# B&R Automation Studio project Parker_BMM_ST_V5_3147_V12 (part 33)

#### nCarriageLR.apt
```
AcoposParameterTable:
  Root Parameters (Disabled=FALSE)
    Configure Parameter (Disabled=FALSE)
      128 = 1 (Name=SGEN_SW_END_IGNORE, Disabled=FALSE)  // Limit values: Ignore SW end positions
      1196 = 0 (Name=PCTRL_MODE_BITS, Disabled=FALSE)  // CTRL Position controller: Mode bits
      90 = 0 (Name=BRAKE_MODE, Disabled=FALSE)  // Motor holding brake: Mode
      80 = 1 (Name=PHASE_MON_IGNORE, Disabled=FALSE)  // Power mains: Ignore phase failure
      390 = 300 (Name=UDC_NOMINAL, Unit=V, Disabled=FALSE)  // CTRL DC bus: Nominal voltage
    VAR_XX_X+0 (Disabled=FALSE)
      777 = VAR_I4_0+0 (Name=FUNCTION_BLOCK_CREATE, Disabled=FALSE)  // VAR_XX_X+0
      VAR_R4_X_0 (Disabled=FALSE)
        4128 = 0.0 (Name=VAR_R4_0+0, Disabled=FALSE)  // velocity set -- cyclic set
        4136 = 0.0 (Name=VAR_R4_1+0, Disabled=FALSE)  // torque limit -- cyclic set
        4144 = 0.736 (Name=VAR_R4_2+0, Disabled=FALSE)  // temp junction Kp
        4152 = 0.736 (Name=VAR_R4_3+0, Disabled=FALSE)  // temp motor Kp
    VAR_XX_X+1 (Disabled=FALSE)
      777 = VAR_I4_0+1 (Name=FUNCTION_BLOCK_CREATE, Disabled=FALSE)  // VAR_XX_X+1
      VAR_R4_X_1 (Disabled=FALSE)
        4129 = 0.0 (Name=VAR_R4_0+1, Disabled=FALSE)  // zero
        4137 = 0.0 (Name=VAR_R4_1+1, Disabled=FALSE)  // 288 - SCTRL_ADD_SET_PARID
        4145 = 0.0 (Name=VAR_R4_2+1, Disabled=FALSE)  // no use
        4153 = 0.0 (Name=VAR_R4_3+1, Disabled=FALSE)  // no use
    VAR_XX_X+2 (Disabled=FALSE)
      777 = VAR_I4_0+2 (Name=FUNCTION_BLOCK_CREATE, Disabled=FALSE)  // VAR_XX_X+2
      VAR_R4_X_2 (Disabled=FALSE)
        4130 = 0.0 (Name=VAR_R4_0+2, Disabled=FALSE)  // Power Consumption Trigger - Left Carriage
        4138 = 0.0 (Name=VAR_R4_1+2, Disabled=FALSE)  // Power Consumption Trigger - Right Carriage
        4146 = 0.0 (Name=VAR_R4_2+2, Disabled=FALSE)  // FB2 FB VAR: Variable2 R4
        4154 = 0.0 (Name=VAR_R4_3+2, Disabled=FALSE)  // FB2 FB VAR: Variable3 R4
    VAR_XX_X+3 (Disabled=FALSE)
      777 = VAR_I4_0+3 (Name=FUNCTION_BLOCK_CREATE, Disabled=FALSE)  // VAR_XX_X+3
      VAR_R4_X_2 (Disabled=FALSE)
        4160 = 0.0 (Name=VAR_I2_0+0, Disabled=FALSE)  // FB0 FB VAR: Variable0 I2
        4168 = 0.0 (Name=VAR_I2_1+0, Disabled=FALSE)  // FB0 FB VAR: Variable1 I2
        4176 = 0.0 (Name=VAR_I2_2+0, Disabled=FALSE)  // FB0 FB VAR: Variable2 I2
        4184 = 0.0 (Name=VAR_I2_3+0, Disabled=FALSE)  // FB0 FB VAR: Variable3 I2
    Velocity Control (Disabled=FALSE)
      Function Create (Disabled=FALSE)
        777 = IPL_MODE+0 (Name=FUNCTION_BLOCK_CREATE, Disabled=FALSE)  // IPL_0
        777 = EVWR_MODE+0 (Name=FUNCTION_BLOCK_CREATE, Disabled=FALSE)  // EVWR_0
        777 = CMP_MODE+0 (Name=FUNCTION_BLOCK_CREATE, Disabled=FALSE)  // CMP_0
        777 = EVWR_MODE+1 (Name=FUNCTION_BLOCK_CREATE, Disabled=FALSE)  // EVWR_1
        777 = ARITH_MODE+6 (Name=FUNCTION_BLOCK_CREATE, Disabled=FALSE)  // EVWR_6
        777 = ARITH_MODE+7 (Name=FUNCTION_BLOCK_CREATE, Disabled=FALSE)  // EVWR_7
      IPL + 0 (Disabled=FALSE)
        8712 = VAR_R4_0+0 (Name=IPL_IN_PARID+0, Disabled=FALSE)  // velocity set
        8760 = CYCLIC_TODRV_COUNT (Name=IPL_EV_PARID+0, Disabled=FALSE)  // 909 - CYCLIC_TODRV_COUNT
        8720 = 2000 (Name=IPL_CYCLE_TIME+0, Unit=us, Disabled=FALSE)  // FB0 FB IPL: Cycle time
        8728 = 800 (Name=IPL_EXTRAPOLATION_TIME+0, Unit=us, Disabled=FALSE)  // FB0 FB IPL: Extrapolation time
        8704 = 1 (Name=IPL_MODE+0, Disabled=FALSE)  // linear interpolation
      EVWR + 0 (Disabled=FALSE)
        4608 = CMP_VALUE+0 (Name=EVWR_EVENT_PARID+0, Disabled=FALSE)  // v_set == 0
        4616 = IPL_VALUE_R4+0 (Name=EVWR_IN_PARID+0, Disabled=FALSE)  // 8752 -- interpolated v_set
        4624 = 0 (Name=EVWR_EVENT_LEVEL+0, Disabled=FALSE)  // FB0 FB EVWR: Event level
        4632 = VAR_R4_1+1 (Name=EVWR_WR_PARID+0, Disabled=FALSE)  // 288 - SCTRL_ADD_SET_PARID
        4640 = 2 (Name=EVWR_MODE+0, Disabled=FALSE)  // cyclic write
      ARITH + 6 (Disabled=FALSE)
        3598 = VCTRL_SCALE_LOAD_UNITS (Name=ARITH_IN1_PARID+6, Disabled=FALSE)  // FB6 FB ARITH: Parameter ID of input1
        3606 = VCTRL_SCALE_LOAD_MOTREV (Name=ARITH_IN2_PARID+6, Disabled=FALSE)  // FB6 FB ARITH: Parameter ID of input2
        3638 = 0 (Name=ARITH_K1+6, Disabled=FALSE)  // FB6 FB ARITH: Multiplication factor1
        3646 = 0 (Name=ARITH_K2+6, Disabled=FALSE)  // FB6 FB ARITH: Multiplication factor2
        3590 = 5 (Name=ARITH_MODE+6, Disabled=FALSE)  // FB6 FB ARITH: Mode
      ARITH + 7 (Disabled=FALSE)
        3599 = VAR_R4_1+1 (Name=ARITH_IN1_PARID+7, Disabled=FALSE)  // FB7 FB ARITH: Parameter ID of input1
        3607 = ARITH_VALUE_R4+6 (Name=ARITH_IN2_PARID+7, Disabled=FALSE)  // FB7 FB ARITH: Parameter ID of input2
        3639 = 0 (Name=ARITH_K1+7, Disabled=FALSE)  // FB7 FB ARITH: Multiplication factor1
        3647 = 0 (Name=ARITH_K2+7, Disabled=FALSE)  // FB7 FB ARITH: Multiplication factor2
        3591 = 5 (Name=ARITH_MODE+7, Disabled=FALSE)  // FB7 FB ARITH: Mode
      288 = ARITH_VALUE_R4+7 (Name=SCTRL_ADD_SET_PARID)  // CTRL Speed controller: Parameter ID additive set value
      CMP + 0 (Disabled=FALSE)
        6656 = IPL_VALUE_R4+0 (Name=CMP_IN_PARID+0, Disabled=FALSE)  // 8752 -- interpolated v_set
        6664 = 0 (Name=CMP_THRESHOLD+0, Disabled=FALSE)  // FB0 FB CMP: threshold
        6672 = 0.001 (Name=CMP_WINDOW+0, Disabled=FALSE)  // FB0 FB CMP: window
        6680 = 0 (Name=CMP_HYSTERESIS+0, Disabled=FALSE)  // FB0 FB CMP: hysteresis window
        6688 = 2 (Name=CMP_MODE+0, Disabled=FALSE)  // ==
      231 = CMP_VALUE+0 (Name=PCTRL_ENABLE_PARID, Disabled=FALSE)  // if(interpolated v_set == 0)enable PCTRL
      EVWR + 1 (Disabled=FALSE)
        4609 = CMP_VALUE+0 (Name=EVWR_EVENT_PARID+1, Disabled=FALSE)  // 6696
        4617 = MOTOR_TORQ_MAX (Name=EVWR_IN_PARID+1, Disabled=FALSE)  // FB1 FB EVWR: Parameter ID of input
        4625 = 1 (Name=EVWR_EVENT_LEVEL+1, Disabled=FALSE)  // FB1 FB EVWR: Event level
        4633 = VAR_R4_1+0 (Name=EVWR_WR_PARID+1, Disabled=FALSE)  // FB1 FB EVWR: Parameter ID of output value
        4641 = 2 (Name=EVWR_MODE+1, Disabled=FALSE)  // mode - cyclic write
    Torque Limitation (Disabled=FALSE)
      Function Create (Disabled=FALSE)
        777 = IPL_MODE+1 (Name=FUNCTION_BLOCK_CREATE, Disabled=FALSE)  // IPL_1
        777 = ARITH_MODE+0 (Name=FUNCTION_BLOCK_CREATE, Disabled=FALSE)  // ARITH_0
        777 = ARITH_MODE+1 (Name=FUNCTION_BLOCK_CREATE, Disabled=FALSE)  // ARITH_1
        777 = ARITH_MODE+2 (Name=FUNCTION_BLOCK_CREATE, Disabled=FALSE)  // ARITH_2
        777 = ARITH_MODE+3 (Name=FUNCTION_BLOCK_CREATE, Disabled=FALSE)  // ARITH_3
        777 = ARITH_MODE+4 (Name=FUNCTION_BLOCK_CREATE, Disabled=FALSE)  // ARITH_4
        777 = ARITH_MODE+5 (Name=FUNCTION_BLOCK_CREATE, Disabled=FALSE)  // ARITH_5
        777 = MINMAX_MODE+0 (Name=FUNCTION_BLOCK_CREATE, Disabled=FALSE)  // MINMAX_0
        777 = MINMAX_MODE+1 (Name=FUNCTION_BLOCK_CREATE, Disabled=FALSE)  // MINMAX_1
        777 = EVWR_MODE+2 (Name=FUNCTION_BLOCK_CREATE, Disabled=FALSE)  // EVWR_2
        777 = EVWR_MODE+3 (Name=FUNCTION_BLOCK_CREATE, Disabled=FALSE)  // EVWR_3
        777 = EVWR_MODE+4 (Name=FUNCTION_BLOCK_CREATE, Disabled=FALSE)  // EVWR_4
        777 = EVWR_MODE+5 (Name=FUNCTION_BLOCK_CREATE, Disabled=FALSE)  // EVWR_5
      IPL (Disabled=FALSE)
        8713 = VAR_R4_1+0 (Name=IPL_IN_PARID+1, Disabled=FALSE)  // 4136
        8761 = CYCLIC_TODRV_COUNT (Name=IPL_EV_PARID+1, Disabled=FALSE)  // 909 - CYCLIC_TODRV_COUNT
        8721 = 2000 (Name=IPL_CYCLE_TIME+1, Unit=us, Disabled=FALSE)  // FB1 FB IPL: Cycle time
        8729 = 2000 (Name=IPL_EXTRAPOLATION_TIME+1, Unit=us, Disabled=FALSE)  // FB1 FB IPL: Extrapolation time
        8705 = 1 (Name=IPL_MODE+1, Disabled=FALSE)  // FB1 FB IPL: Mode -- linear interpolation
      ARITH + 0 (Disabled=FALSE)
        3592 = TEMP_JUNCTION_LIM (Name=ARITH_IN1_PARID+0, Disabled=FALSE)  // TEMP_JUNCTION_LIM -- 842
        3600 = TEMP_JUNCTION (Name=ARITH_IN2_PARID+0, Disabled=FALSE)  // TEMP_JUNCTION -- 382
        3632 = 0 (Name=ARITH_K1+0, Disabled=FALSE)  // FB0 FB ARITH: Multiplication factor1
        3640 = 0 (Name=ARITH_K2+0, Disabled=FALSE)  // FB0 FB ARITH: Multiplication factor2
        3584 = 2 (Name=ARITH_MODE+0, Disabled=FALSE)  // y= x1 - x2
      ARITH + 1 (Disabled=FALSE)
        3593 = ARITH_VALUE_R4+0 (Name=ARITH_IN1_PARID+1, Disabled=FALSE)  // 3624
        3601 = VAR_R4_2+0 (Name=ARITH_IN2_PARID+1, Disabled=FALSE)  // 4144
        3633 = 0 (Name=ARITH_K1+1, Disabled=FALSE)  // FB1 FB ARITH: Multiplication factor1
        3641 = 0 (Name=ARITH_K2+1, Disabled=FALSE)  // FB1 FB ARITH: Multiplication factor2
        3585 = 3 (Name=ARITH_MODE+1, Disabled=FALSE)  // y = x1 * x2
      ARITH + 2 (Disabled=FALSE)
        3594 = MOTOR_TORQ_RATED (Name=ARITH_IN1_PARID+2, Disabled=FALSE)  // MOTOR_TORQ_RATED -- 53
        3602 = ARITH_VALUE_R4+1 (Name=ARITH_IN2_PARID+2, Disabled=FALSE)  // 3625
        3634 = 0 (Name=ARITH_K1+2, Disabled=FALSE)  // FB2 FB ARITH: Multiplication factor1
        3642 = 0 (Name=ARITH_K2+2, Disabled=FALSE)  // FB2 FB ARITH: Multiplication factor2
        3586 = 1 (Name=ARITH_MODE+2, Disabled=FALSE)  // y = x1 + x2
      ARITH + 3 (Disabled=FALSE)
        3595 = MOTOR_WIND_TEMP_MAX (Name=ARITH_IN1_PARID+3, Disabled=FALSE)  // 74 - MOTOR_WIND_TEMP_MAX
        3603 = TEMP_MOTOR_MODELL (Name=ARITH_IN2_PARID+3, Disabled=FALSE)  // 393 - TEMP_MOTOR_MODELL
        3635 = 0 (Name=ARITH_K1+3, Disabled=FALSE)  // FB3 FB ARITH: Multiplication factor1
        3643 = 0 (Name=ARITH_K2+3, Disabled=FALSE)  // FB3 FB ARITH: Multiplication factor2
        3587 = 2 (Name=ARITH_MODE+3, Disabled=FALSE)  // y = x1 - x2
      ARITH + 4 (Disabled=FALSE)
        3596 = ARITH_VALUE_R4+3 (Name=ARITH_IN1_PARID+4, Disabled=FALSE)  // 3627
        3604 = VAR_R4_3+0 (Name=ARITH_IN2_PARID+4, Disabled=FALSE)  // 4152
        3636 = 0 (Name=ARITH_K1+4, Disabled=FALSE)  // FB4 FB ARITH: Multiplication factor1
        3644 = 0 (Name=ARITH_K2+4, Disabled=FALSE)  // FB4 FB ARITH: Multiplication factor2
        3588 = 3 (Name=ARITH_MODE+4, Disabled=FALSE)  // y = x1 * x2
      ARITH + 5 (Disabled=FALSE)
        3597 = MOTOR_TORQ_RATED (Name=ARITH_IN1_PARID+5, Disabled=FALSE)  // MOTOR_TORQ_RATED -- 53
        3605 = ARITH_VALUE_R4+4 (Name=ARITH_IN2_PARID+5, Disabled=FALSE)  // 3628
        3637 = 0 (Name=ARITH_K1+5, Disabled=FALSE)  // FB5 FB ARITH: Multiplication factor1
        3645 = 0 (Name=ARITH_K2+5, Disabled=FALSE)  // FB5 FB ARITH: Multiplication factor2
        3589 = 1 (Name=ARITH_MODE+5, Disabled=FALSE)  // y = x1 + x2
      MINMAX + 0 (Disabled=FALSE)
        12312 = MOTOR_TORQ_MAX (Name=MINMAX_IN1_PARID+0, Disabled=FALSE)  // MOTOR_TORQ_MAX -- 54
        12320 = ARITH_VALUE_R4+2 (Name=MINMAX_IN2_PARID+0, Disabled=FALSE)  // 3626
        12328 = ARITH_VALUE_R4+5 (Name=MINMAX_IN3_PARID+0, Disabled=FALSE)  // 3629
        12336 = IPL_VALUE_R4+1 (Name=MINMAX_IN4_PARID+0, Disabled=FALSE)  // 8753 -- interpolated torque set
        12288 = 1 (Name=MINMAX_MODE+0, Disabled=FALSE)  // MIN(MOTOR_TORQ_MAX,ARITH_VALUE_R4+1)
      MINMAX + 1 (Disabled=FALSE)
        12313 = VAR_R4_0+1 (Name=MINMAX_IN1_PARID+1, Disabled=FALSE)  // zero
        12321 = MINMAX_VALUE_R4+0 (Name=MINMAX_IN2_PARID+1, Disabled=FALSE)  // FB1 FB MINMAX: Parameter ID of input2
        12289 = 2 (Name=MINMAX_MODE+1, Disabled=FALSE)  // MAX(VAR_R4_0+1,MINMAX_VALUE_R4+0)
      EVWR + 2 (Disabled=FALSE)
        4610 = CONST_I4_ONE (Name=EVWR_EVENT_PARID+2, Disabled=FALSE)  // FB2 FB EVWR: Parameter ID of event input
        4618 = MINMAX_VALUE_R4+1 (Name=EVWR_IN_PARID+2, Disabled=FALSE)  // FB2 FB EVWR: Parameter ID of input
        4626 = 1 (Name=EVWR_EVENT_LEVEL+2, Disabled=FALSE)  // FB2 FB EVWR: Event level
        4634 = LIM_T2_POS (Name=EVWR_WR_PARID+2, Disabled=FALSE)  // 348
        4642 = 2 (Name=EVWR_MODE+2, Disabled=FALSE)  // mode - cyclic write
      EVWR + 3 (Disabled=FALSE)
        4611 = CONST_I4_ONE (Name=EVWR_EVENT_PARID+3, Disabled=FALSE)  // FB3 FB EVWR: Parameter ID of event input
        4619 = MINMAX_VALUE_R4+1 (Name=EVWR_IN_PARID+3, Disabled=FALSE)  // FB3 FB EVWR: Parameter ID of input
        4627 = 1 (Name=EVWR_EVENT_LEVEL+3, Disabled=FALSE)  // FB3 FB EVWR: Event level
        4635 = LIM_T2_NEG (Name=EVWR_WR_PARID+3, Disabled=FALSE)  // 349
        4643 = 2 (Name=EVWR_MODE+3, Disabled=FALSE)  // mode - cyclic write
      EVWR + 4 (Disabled=FALSE)
        4612 = CONST_I4_ONE (Name=EVWR_EVENT_PARID+4, Disabled=FALSE)  // FB4 FB EVWR: Parameter ID of event input
        4620 = MINMAX_VALUE_R4+1 (Name=EVWR_IN_PARID+4, Disabled=FALSE)  // FB4 FB EVWR: Parameter ID of input
        4628 = 1 (Name=EVWR_EVENT_LEVEL+4, Disabled=FALSE)  // FB4 FB EVWR: Event level
        4636 = LIM_T1_POS (Name=EVWR_WR_PARID+4, Disabled=FALSE)  // 248
        4644 = 2 (Name=EVWR_MODE+4, Disabled=FALSE)  // mode - cyclic write
      EVWR + 5 (Disabled=FALSE)
        4613 = CONST_I4_ONE (Name=EVWR_EVENT_PARID+5, Disabled=FALSE)  // FB5 FB EVWR: Parameter ID of event input
        4621 = MINMAX_VALUE_R4+1 (Name=EVWR_IN_PARID+5, Disabled=FALSE)  // FB5 FB EVWR: Parameter ID of input
        4629 = 1 (Name=EVWR_EVENT_LEVEL+5, Disabled=FALSE)  // FB5 FB EVWR: Event level
        4637 = LIM_T1_NEG (Name=EVWR_WR_PARID+5, Disabled=FALSE)  // 249
        4645 = 2 (Name=EVWR_MODE+5, Disabled=FALSE)  // mode - cyclic write
    brake resistors (Disabled=TRUE)
      10 = 33 (Name=R_BLEEDER_EXT, Unit=Ohm, Disabled=TRUE)  // Bleeder: External: Resistance
      11 = 637 (Name=TEMP_MAX_BLEEDER_EXT, Unit=°C, Disabled=TRUE)  // Bleeder: External: Limit temperature
      12 = 0.852 (Name=RTH_BLEEDER_AMB_EXT, Unit=K/W, Disabled=TRUE)  // Bleeder: External: Thermal resistance
      13 = 40.68 (Name=CTH_BLEEDER_EXT, Unit=Ws/K, Disabled=TRUE)  // Bleeder: External: Thermal capacity
      398 = 1 (Name=BLEEDER_SELECTOR_EXT, Disabled=TRUE)  // Bleeder: Selector
    8B0W0079H000.000-1 mounting vertical V1 (Disabled=TRUE)
      brake  (Disabled=TRUE)  //  DO NOT USE with ACOPOS Firmware before V2.27.0
      10 = 33 (Name=R_BLEEDER_EXT, Unit=Ohm, Disabled=TRUE)  // Bleeder: External: Resistance
      11 = 673.08 (Name=TEMP_MAX_BLEEDER_EXT, Unit=癈, Disabled=TRUE)  // Bleeder: External: Limit temperature
      12 = 0.852 (Name=RTH_BLEEDER_AMB_EXT, Unit=K/W, Disabled=TRUE)  // Bleeder: External: Thermic resistance
      13 = 40.68 (Name=CTH_BLEEDER_EXT, Unit=Ws/K, Disabled=TRUE)  // Bleeder: External: Thermic capacity
      398 = 1 (Name=BLEEDER_SELECTOR_EXT, Disabled=TRUE)  // Bleeder: Selector
    Power Consumption (Disabled=TRUE)
      1140 = 10000000 (Name=PMET_TIME_IV, Unit=us, Disabled=TRUE)  // PowerMeter: Observation period
      1139 = 1 (Name=PMET_MODE, Disabled=TRUE)  // PowerMeter: Mode
    HardWare Limit  For ACOPOS Multi:
      945 = VAR_I2_0+0 (Name=POS_LIMIT_SWITCH_PARID)  // Digital inputs: Parameter ID for positive end switch
      946 = VAR_I2_1+0 (Name=NEG_LIMIT_SWITCH_PARID)  // Digital inputs: Parameter ID for negative end switch
```

### Data object Logical/Motion/para/BlowPin2LR (Apt)

#### BlowPin2LR.apt
```
AcoposParameterTable:
  Root Parameters (Disabled=FALSE)
    Configure Parameter (Disabled=FALSE)
      128 = 1 (Name=SGEN_SW_END_IGNORE, Disabled=FALSE)  // Limit values: Ignore SW end positions
      1196 = 0 (Name=PCTRL_MODE_BITS, Disabled=FALSE)  // CTRL Position controller: Mode bits
      80 = 1 (Name=PHASE_MON_IGNORE, Disabled=TRUE)  // Power mains: Ignore phase failure
      300 = 311 (Name=UDC_DETECTION, Unit=V, Disabled=FALSE)  // CTRL DC bus: Voltage detection: Lower limit
      373 = 1 (Name=TEMP_MOTOR_MODEL_MODE)  // Motor: Temperature model: Mode
      1215 = 2 (Name=MOTOR_TEMPSENS_TYPE, Disabled=TRUE)  // Temperature sensor: Type
    VAR_XX_X+0 (Disabled=FALSE)
      777 = VAR_I4_0+0 (Name=FUNCTION_BLOCK_CREATE, Disabled=FALSE)  // VAR_XX_X+0
      VAR_R4_X_0 (Disabled=FALSE)
        4128 = 0.0 (Name=VAR_R4_0+0, Disabled=FALSE)  // velocity set -- cyclic set
        4136 = 0.0 (Name=VAR_R4_1+0, Disabled=FALSE)  // torque limit -- cyclic set
        4144 = 0.666 (Name=VAR_R4_2+0, Disabled=FALSE)  // temp junction Kp
        4152 = 0.666 (Name=VAR_R4_3+0, Disabled=FALSE)  // temp motor Kp
    VAR_XX_X+1 (Disabled=FALSE)
      777 = VAR_I4_0+1 (Name=FUNCTION_BLOCK_CREATE, Disabled=FALSE)  // VAR_XX_X+1
      VAR_R4_X_1 (Disabled=FALSE)
        4129 = 0.0 (Name=VAR_R4_0+1, Disabled=FALSE)  // zero
        4137 = 0.0 (Name=VAR_R4_1+1, Disabled=FALSE)  // 288 - SCTRL_ADD_SET_PARID
        4145 = 0.0 (Name=VAR_R4_2+1, Disabled=FALSE)  // no use
        4153 = 0.0 (Name=VAR_R4_3+1, Disabled=FALSE)  // no use
    VAR_XX_X+3 (Disabled=FALSE)
      777 = VAR_I4_0+3 (Name=FUNCTION_BLOCK_CREATE, Disabled=FALSE)  // VAR_XX_X+3
      VAR_R4_X_2 (Disabled=FALSE)
        4160 = 0.0 (Name=VAR_I2_0+0, Disabled=FALSE)  // FB0 FB VAR: Variable0 I2
        4168 = 0.0 (Name=VAR_I2_1+0, Disabled=FALSE)  // FB0 FB VAR: Variable1 I2
        4176 = 0.0 (Name=VAR_I2_2+0, Disabled=FALSE)  // FB0 FB VAR: Variable2 I2
        4184 = 0.0 (Name=VAR_I2_3+0, Disabled=FALSE)  // FB0 FB VAR: Variable3 I2
    Velocity Control (Disabled=FALSE)
      Function Create (Disabled=FALSE)
        777 = IPL_MODE+0 (Name=FUNCTION_BLOCK_CREATE, Disabled=FALSE)  // IPL_0
        777 = EVWR_MODE+0 (Name=FUNCTION_BLOCK_CREATE, Disabled=FALSE)  // EVWR_0
        777 = CMP_MODE+0 (Name=FUNCTION_BLOCK_CREATE, Disabled=FALSE)  // CMP_0
        777 = EVWR_MODE+1 (Name=FUNCTION_BLOCK_CREATE, Disabled=FALSE)  // EVWR_1
      IPL + 0 (Disabled=FALSE)
        8712 = VAR_R4_0+0 (Name=IPL_IN_PARID+0, Disabled=FALSE)  // velocity set
        8760 = CYCLIC_TODRV_COUNT (Name=IPL_EV_PARID+0, Disabled=FALSE)  // 909 - CYCLIC_TODRV_COUNT
        8720 = 2000 (Name=IPL_CYCLE_TIME+0, Unit=us, Disabled=FALSE)  // FB0 FB IPL: Cycle time
        8728 = 800 (Name=IPL_EXTRAPOLATION_TIME+0, Unit=us, Disabled=FALSE)  // FB0 FB IPL: Extrapolation time
        8704 = 1 (Name=IPL_MODE+0, Disabled=FALSE)  // linear interpolation
      EVWR + 0 (Disabled=FALSE)
        4608 = CMP_VALUE+0 (Name=EVWR_EVENT_PARID+0, Disabled=FALSE)  // v_set == 0
        4616 = IPL_VALUE_R4+0 (Name=EVWR_IN_PARID+0, Disabled=FALSE)  // 8752 -- interpolated v_set
        4624 = 0 (Name=EVWR_EVENT_LEVEL+0, Disabled=FALSE)  // FB0 FB EVWR: Event level
        4632 = VAR_R4_1+1 (Name=EVWR_WR_PARID+0, Disabled=FALSE)  // 288-SCTRL_ADD_SET_PARID
        4640 = 2 (Name=EVWR_MODE+0, Disabled=FALSE)  // cyclic write
      288 = VAR_R4_1+1 (Name=SCTRL_ADD_SET_PARID, Disabled=FALSE)  // CTRL Speed controller: Parameter ID additive set value
      CMP + 0 (Disabled=FALSE)
        6656 = IPL_VALUE_R4+0 (Name=CMP_IN_PARID+0, Disabled=FALSE)  // 8752 -- interpolated v_set
        6664 = 0 (Name=CMP_THRESHOLD+0, Disabled=FALSE)  // FB0 FB CMP: threshold
        6672 = 0.001 (Name=CMP_WINDOW+0, Disabled=FALSE)  // FB0 FB CMP: window
        6680 = 0 (Name=CMP_HYSTERESIS+0, Disabled=FALSE)  // FB0 FB CMP: hysteresis window
        6688 = 2 (Name=CMP_MODE+0, Disabled=FALSE)  // ==
      231 = CMP_VALUE+0 (Name=PCTRL_ENABLE_PARID, Disabled=FALSE)  // if(interpolated v_set == 0)enable PCTRL
      EVWR + 1 (Disabled=FALSE)
        4609 = CMP_VALUE+0 (Name=EVWR_EVENT_PARID+1, Disabled=FALSE)  // 6696
        4617 = MOTOR_TORQ_MAX (Name=EVWR_IN_PARID+1, Disabled=FALSE)  // FB1 FB EVWR: Parameter ID of input
        4625 = 1 (Name=EVWR_EVENT_LEVEL+1, Disabled=FALSE)  // FB1 FB EVWR: Event level
        4633 = VAR_R4_1+0 (Name=EVWR_WR_PARID+1, Disabled=FALSE)  // FB1 FB EVWR: Parameter ID of output value
        4641 = 2 (Name=EVWR_MODE+1, Disabled=FALSE)  // mode - cyclic write
    Torque Limitation (Disabled=FALSE)
      Function Create (Disabled=FALSE)
        777 = IPL_MODE+1 (Name=FUNCTION_BLOCK_CREATE, Disabled=FALSE)  // IPL_1
        777 = ARITH_MODE+0 (Name=FUNCTION_BLOCK_CREATE, Disabled=FALSE)  // ARITH_0
        777 = ARITH_MODE+1 (Name=FUNCTION_BLOCK_CREATE, Disabled=FALSE)  // ARITH_1
        777 = ARITH_MODE+2 (Name=FUNCTION_BLOCK_CREATE, Disabled=FALSE)  // ARITH_2
        777 = ARITH_MODE+3 (Name=FUNCTION_BLOCK_CREATE, Disabled=FALSE)  // ARITH_3
        777 = ARITH_MODE+4 (Name=FUNCTION_BLOCK_CREATE, Disabled=FALSE)  // ARITH_4
        777 = ARITH_MODE+5 (Name=FUNCTION_BLOCK_CREATE, Disabled=FALSE)  // ARITH_5
        777 = MINMAX_MODE+0 (Name=FUNCTION_BLOCK_CREATE, Disabled=FALSE)  // MINMAX_0
        777 = MINMAX_MODE+1 (Name=FUNCTION_BLOCK_CREATE, Disabled=FALSE)  // MINMAX_1
        777 = EVWR_MODE+2 (Name=FUNCTION_BLOCK_CREATE, Disabled=FALSE)  // EVWR_2
        777 = EVWR_MODE+3 (Name=FUNCTION_BLOCK_CREATE, Disabled=FALSE)  // EVWR_3
        777 = EVWR_MODE+4 (Name=FUNCTION_BLOCK_CREATE, Disabled=FALSE)  // EVWR_4
        777 = EVWR_MODE+5 (Name=FUNCTION_BLOCK_CREATE, Disabled=FALSE)  // EVWR_5
      IPL (Disabled=FALSE)
        8713 = VAR_R4_1+0 (Name=IPL_IN_PARID+1, Disabled=FALSE)  // 4136
        8761 = CYCLIC_TODRV_COUNT (Name=IPL_EV_PARID+1, Disabled=FALSE)  // 909 - CYCLIC_TODRV_COUNT
        8721 = 2000 (Name=IPL_CYCLE_TIME+1, Unit=us, Disabled=FALSE)  // FB1 FB IPL: Cycle time
        8729 = 2000 (Name=IPL_EXTRAPOLATION_TIME+1, Unit=us, Disabled=FALSE)  // FB1 FB IPL: Extrapolation time
        8705 = 1 (Name=IPL_MODE+1, Disabled=FALSE)  // FB1 FB IPL: Mode -- linear interpolation
      ARITH + 0 (Disabled=FALSE)
        3592 = TEMP_JUNCTION_LIM (Name=ARITH_IN1_PARID+0, Disabled=FALSE)  // TEMP_JUNCTION_LIM -- 842
        3600 = TEMP_JUNCTION (Name=ARITH_IN2_PARID+0, Disabled=FALSE)  // TEMP_JUNCTION -- 382
        3632 = 0 (Name=ARITH_K1+0, Disabled=FALSE)  // FB0 FB ARITH: Multiplication factor1
        3640 = 0 (Name=ARITH_K2+0, Disabled=FALSE)  // FB0 FB ARITH: Multiplication factor2
        3584 = 2 (Name=ARITH_MODE+0, Disabled=FALSE)  // y= x1 - x2
      ARITH + 1 (Disabled=FALSE)
        3593 = ARITH_VALUE_R4+0 (Name=ARITH_IN1_PARID+1, Disabled=FALSE)  // 3624
        3601 = VAR_R4_2+0 (Name=ARITH_IN2_PARID+1, Disabled=FALSE)  // 4144
        3633 = 0 (Name=ARITH_K1+1, Disabled=FALSE)  // FB1 FB ARITH: Multiplication factor1
        3641 = 0 (Name=ARITH_K2+1, Disabled=FALSE)  // FB1 FB ARITH: Multiplication factor2
        3585 = 3 (Name=ARITH_MODE+1, Disabled=FALSE)  // y = x1 * x2
      ARITH + 2 (Disabled=FALSE)
        3594 = MOTOR_TORQ_RATED (Name=ARITH_IN1_PARID+2, Disabled=FALSE)  // MOTOR_TORQ_RATED -- 53
        3602 = ARITH_VALUE_R4+1 (Name=ARITH_IN2_PARID+2, Disabled=FALSE)  // 3625
        3634 = 0 (Name=ARITH_K1+2, Disabled=FALSE)  // FB2 FB ARITH: Multiplication factor1
        3642 = 0 (Name=ARITH_K2+2, Disabled=FALSE)  // FB2 FB ARITH: Multiplication factor2
        3586 = 1 (Name=ARITH_MODE+2, Disabled=FALSE)  // y = x1 + x2
      ARITH + 3 (Disabled=FALSE)
        3595 = MOTOR_WIND_TEMP_MAX (Name=ARITH_IN1_PARID+3, Disabled=FALSE)  // 74 - MOTOR_WIND_TEMP_MAX
        3603 = TEMP_MOTOR_MODELL (Name=ARITH_IN2_PARID+3, Disabled=FALSE)  // 393 - TEMP_MOTOR_MODELL
        3635 = 0 (Name=ARITH_K1+3, Disabled=FALSE)  // FB3 FB ARITH: Multiplication factor1
        3643 = 0 (Name=ARITH_K2+3, Disabled=FALSE)  // FB3 FB ARITH: Multiplication factor2
        3587 = 2 (Name=ARITH_MODE+3, Disabled=FALSE)  // y = x1 - x2
      ARITH + 4 (Disabled=FALSE)
        3596 = ARITH_VALUE_R4+3 (Name=ARITH_IN1_PARID+4, Disabled=FALSE)  // 3627
        3604 = VAR_R4_3+0 (Name=ARITH_IN2_PARID+4, Disabled=FALSE)  // 4152
        3636 = 0 (Name=ARITH_K1+4, Disabled=FALSE)  // FB4 FB ARITH: Multiplication factor1
        3644 = 0 (Name=ARITH_K2+4, Disabled=FALSE)  // FB4 FB ARITH: Multiplication factor2
        3588 = 3 (Name=ARITH_MODE+4, Disabled=FALSE)  // y = x1 * x2
      ARITH + 5 (Disabled=FALSE)
        3597 = MOTOR_TORQ_RATED (Name=ARITH_IN1_PARID+5, Disabled=FALSE)  // MOTOR_TORQ_RATED -- 53
        3605 = ARITH_VALUE_R4+4 (Name=ARITH_IN2_PARID+5, Disabled=FALSE)  // 3628
        3637 = 0 (Name=ARITH_K1+5, Disabled=FALSE)  // FB5 FB ARITH: Multiplication factor1
        3645 = 0 (Name=ARITH_K2+5, Disabled=FALSE)  // FB5 FB ARITH: Multiplication factor2
        3589 = 1 (Name=ARITH_MODE+5, Disabled=FALSE)  // y = x1 + x2
      MINMAX + 0 (Disabled=FALSE)
        12312 = MOTOR_TORQ_MAX (Name=MINMAX_IN1_PARID+0, Disabled=FALSE)  // MOTOR_TORQ_MAX -- 54
        12320 = ARITH_VALUE_R4+2 (Name=MINMAX_IN2_PARID+0, Disabled=FALSE)  // 3626
        12328 = ARITH_VALUE_R4+5 (Name=MINMAX_IN3_PARID+0, Disabled=FALSE)  // 3629
        12336 = IPL_VALUE_R4+1 (Name=MINMAX_IN4_PARID+0, Disabled=FALSE)  // 8753 -- interpolated torque set
        12288 = 1 (Name=MINMAX_MODE+0, Disabled=FALSE)  // MIN(MOTOR_TORQ_MAX,ARITH_VALUE_R4+1)
      MINMAX + 1 (Disabled=FALSE)
        12313 = VAR_R4_0+1 (Name=MINMAX_IN1_PARID+1, Disabled=FALSE)  // zero
        12321 = MINMAX_VALUE_R4+0 (Name=MINMAX_IN2_PARID+1, Disabled=FALSE)  // FB1 FB MINMAX: Parameter ID of input2
        12289 = 2 (Name=MINMAX_MODE+1, Disabled=FALSE)  // MAX(VAR_R4_0+1,MINMAX_VALUE_R4+0)
      EVWR + 2 (Disabled=FALSE)
        4610 = CONST_I4_ONE (Name=EVWR_EVENT_PARID+2, Disabled=FALSE)  // FB2 FB EVWR: Parameter ID of event input
        4618 = MINMAX_VALUE_R4+1 (Name=EVWR_IN_PARID+2, Disabled=FALSE)  // FB2 FB EVWR: Parameter ID of input
        4626 = 1 (Name=EVWR_EVENT_LEVEL+2, Disabled=FALSE)  // FB2 FB EVWR: Event level
        4634 = LIM_T2_POS (Name=EVWR_WR_PARID+2, Disabled=FALSE)  // 348
        4642 = 2 (Name=EVWR_MODE+2, Disabled=FALSE)  // mode - cyclic write
      EVWR + 3 (Disabled=FALSE)
        4611 = CONST_I4_ONE (Name=EVWR_EVENT_PARID+3, Disabled=FALSE)  // FB3 FB EVWR: Parameter ID of event input
        4619 = MINMAX_VALUE_R4+1 (Name=EVWR_IN_PARID+3, Disabled=FALSE)  // FB3 FB EVWR: Parameter ID of input
        4627 = 1 (Name=EVWR_EVENT_LEVEL+3, Disabled=FALSE)  // FB3 FB EVWR: Event level
        4635 = LIM_T2_NEG (Name=EVWR_WR_PARID+3, Disabled=FALSE)  // 349
        4643 = 2 (Name=EVWR_MODE+3, Disabled=FALSE)  // mode - cyclic write
      EVWR + 4 (Disabled=FALSE)
        4612 = CONST_I4_ONE (Name=EVWR_EVENT_PARID+4, Disabled=FALSE)  // FB4 FB EVWR: Parameter ID of event input
        4620 = MINMAX_VALUE_R4+1 (Name=EVWR_IN_PARID+4, Disabled=FALSE)  // FB4 FB EVWR: Parameter ID of input
        4628 = 1 (Name=EVWR_EVENT_LEVEL+4, Disabled=FALSE)  // FB4 FB EVWR: Event level
        4636 = LIM_T1_POS (Name=EVWR_WR_PARID+4, Disabled=FALSE)  // 248
        4644 = 2 (Name=EVWR_MODE+4, Disabled=FALSE)  // mode - cyclic write
      EVWR + 5 (Disabled=FALSE)
        4613 = CONST_I4_ONE (Name=EVWR_EVENT_PARID+5, Disabled=FALSE)  // FB5 FB EVWR: Parameter ID of event input
        4621 = MINMAX_VALUE_R4+1 (Name=EVWR_IN_PARID+5, Disabled=FALSE)  // FB5 FB EVWR: Parameter ID of input
        4629 = 1 (Name=EVWR_EVENT_LEVEL+5, Disabled=FALSE)  // FB5 FB EVWR: Event level
        4637 = LIM_T1_NEG (Name=EVWR_WR_PARID+5, Disabled=FALSE)  // 249
        4645 = 2 (Name=EVWR_MODE+5, Disabled=FALSE)  // mode - cyclic write
    HardWare Limit  For ACOPOS Multi:
      945 = VAR_I2_0+0 (Name=POS_LIMIT_SWITCH_PARID)  // Digital inputs: Parameter ID for positive end switch
      946 = VAR_I2_1+0 (Name=NEG_LIMIT_SWITCH_PARID)  // Digital inputs: Parameter ID for negative end switch
```

### Data object Logical/Motion/para/ClampLR (Apt)

#### ClampLR.apt
```
AcoposParameterTable:
  Root Parameters (Disabled=FALSE)
    Configure Parameter (Disabled=FALSE)
      128 = 1 (Name=SGEN_SW_END_IGNORE, Disabled=FALSE)  // Limit values: Ignore SW end positions
      1196 = 0 (Name=PCTRL_MODE_BITS, Disabled=FALSE)  // CTRL Position controller: Mode bits
      80 = 1 (Name=PHASE_MON_IGNORE, Disabled=FALSE)  // Power mains: Ignore phase failure
      300 = 300 (Name=UDC_DETECTION, Unit=V, Disabled=FALSE)  // CTRL DC bus: Voltage detection: Lower limit
      373 = 0 (Name=TEMP_MOTOR_MODEL_MODE)  // Motor: Temperature model: Mode
    VAR_XX_X+0 (Disabled=FALSE)
      777 = VAR_I4_0+0 (Name=FUNCTION_BLOCK_CREATE, Disabled=FALSE)  // VAR_XX_X+0
      VAR_R4_X_0 (Disabled=FALSE)
        4128 = 0.0 (Name=VAR_R4_0+0, Disabled=FALSE)  // velocity set -- cyclic set
        4136 = 0.0 (Name=VAR_R4_1+0, Disabled=FALSE)  // torque limit -- cyclic set
        4144 = 3.226 (Name=VAR_R4_2+0, Disabled=FALSE)  // temp junction Kp : (Peak - nominal)/50  (205-43.7)/50
        4152 = 3.226 (Name=VAR_R4_3+0, Disabled=FALSE)  // temp motor Kp
      VAR_I4_X_0 (Disabled=FALSE)
        4160 = 0.0 (Name=VAR_I2_0+0, Disabled=FALSE)  // FB0 FB VAR: Variable0 I2
        4168 = 0.0 (Name=VAR_I2_1+0, Disabled=FALSE)  // FB0 FB VAR: Variable1 I2
        4176 = 0.0 (Name=VAR_I2_2+0, Disabled=FALSE)  // FB0 FB VAR: Variable2 I2
        4184 = 0.0 (Name=VAR_I2_3+0, Disabled=FALSE)  // FB0 FB VAR: Variable3 I2
    VAR_XX_X+1 (Disabled=FALSE)
      777 = VAR_I4_0+1 (Name=FUNCTION_BLOCK_CREATE, Disabled=FALSE)  // VAR_XX_X+1
      VAR_R4_X_1 (Disabled=FALSE)
        4129 = 0.0 (Name=VAR_R4_0+1, Disabled=FALSE)  // zero
        4137 = 0.0 (Name=VAR_R4_1+1, Disabled=FALSE)  // 288 - SCTRL_ADD_SET_PARID
        4145 = 104 (Name=VAR_R4_2+1, Disabled=FALSE)  // Torque_Max - User Setting
        4153 = 0.0 (Name=VAR_R4_3+1, Disabled=FALSE)  // no use
    VAR_XX_X+2 (Disabled=FALSE)
      777 = VAR_I4_0+2 (Name=FUNCTION_BLOCK_CREATE, Disabled=FALSE)  // VAR_XX_X+2
      VAR_R4_X_2 (Disabled=FALSE)
        4130 = 0.0 (Name=VAR_R4_0+2, Disabled=FALSE)  // Power Consumption Trigger - Left Carriage
        4138 = 0.0 (Name=VAR_R4_1+2, Disabled=FALSE)  // Power Consumption Trigger - Right Carriage
        4146 = 0.0 (Name=VAR_R4_2+2, Disabled=FALSE)  // FB2 FB VAR: Variable2 R4
        4154 = 0.0 (Name=VAR_R4_3+2, Disabled=FALSE)  // FB2 FB VAR: Variable3 R4
    Velocity Control (Disabled=FALSE)
      Function Create (Disabled=FALSE)
        777 = IPL_MODE+0 (Name=FUNCTION_BLOCK_CREATE, Disabled=FALSE)  // IPL_0
        777 = EVWR_MODE+0 (Name=FUNCTION_BLOCK_CREATE, Disabled=FALSE)  // EVWR_0
        777 = CMP_MODE+0 (Name=FUNCTION_BLOCK_CREATE, Disabled=FALSE)  // CMP_0
        777 = EVWR_MODE+1 (Name=FUNCTION_BLOCK_CREATE, Disabled=FALSE)  // EVWR_1
      IPL + 0 (Disabled=FALSE)
        8712 = VAR_R4_0+0 (Name=IPL_IN_PARID+0, Disabled=FALSE)  // velocity set
        8760 = CYCLIC_TODRV_COUNT (Name=IPL_EV_PARID+0, Disabled=FALSE)  // 909 - CYCLIC_TODRV_COUNT
        8720 = 2000 (Name=IPL_CYCLE_TIME+0, Unit=us, Disabled=FALSE)  // FB0 FB IPL: Cycle time
        8728 = 800 (Name=IPL_EXTRAPOLATION_TIME+0, Unit=us, Disabled=FALSE)  // FB0 FB IPL: Extrapolation time
        8704 = 1 (Name=IPL_MODE+0, Disabled=FALSE)  // linear interpolation
      EVWR + 0 (Disabled=FALSE)
        4608 = CMP_VALUE+0 (Name=EVWR_EVENT_PARID+0, Disabled=FALSE)  // v_set == 0
        4616 = IPL_VALUE_R4+0 (Name=EVWR_IN_PARID+0, Disabled=FALSE)  // 8752 -- interpolated v_set
        4624 = 0 (Name=EVWR_EVENT_LEVEL+0, Disabled=FALSE)  // FB0 FB EVWR: Event level
        4632 = VAR_R4_1+1 (Name=EVWR_WR_PARID+0, Disabled=FALSE)  // 288 - SCTRL_ADD_SET_PARID
        4640 = 2 (Name=EVWR_MODE+0, Disabled=FALSE)  // cyclic write
      288 = VAR_R4_1+1 (Name=SCTRL_ADD_SET_PARID, Disabled=FALSE)  // CTRL Speed controller: Parameter ID additive set value
      CMP + 0 (Disabled=FALSE)
        6656 = IPL_VALUE_R4+0 (Name=CMP_IN_PARID+0, Disabled=FALSE)  // 8752 -- interpolated v_set
        6664 = 0 (Name=CMP_THRESHOLD+0, Disabled=FALSE)  // FB0 FB CMP: threshold
        6672 = 0.001 (Name=CMP_WINDOW+0, Disabled=FALSE)  // FB0 FB CMP: window
        6680 = 0 (Name=CMP_HYSTERESIS+0, Disabled=FALSE)  // FB0 FB CMP: hysteresis window
        6688 = 2 (Name=CMP_MODE+0, Disabled=FALSE)  // ==
      231 = CMP_VALUE+0 (Name=PCTRL_ENABLE_PARID, Disabled=FALSE)  // if(interpolated v_set == 0)enable PCTRL
      EVWR + 1 (Disabled=FALSE)
        4609 = CMP_VALUE+0 (Name=EVWR_EVENT_PARID+1, Disabled=FALSE)  // 6696
        4617 = VAR_R4_2+1 (Name=EVWR_IN_PARID+1, Disabled=FALSE)  // FB1 FB EVWR: Parameter ID of input / Torque_Max - User Setting
        4625 = 1 (Name=EVWR_EVENT_LEVEL+1, Disabled=FALSE)  // FB1 FB EVWR: Event level
        4633 = VAR_R4_1+0 (Name=EVWR_WR_PARID+1, Disabled=FALSE)  // FB1 FB EVWR: Parameter ID of output value
        4641 = 2 (Name=EVWR_MODE+1, Disabled=FALSE)  // mode - cyclic write
    Torque Limitation (Disabled=FALSE)
      Function Create (Disabled=FALSE)
        777 = IPL_MODE+1 (Name=FUNCTION_BLOCK_CREATE, Disabled=FALSE)  // IPL_1
        777 = ARITH_MODE+0 (Name=FUNCTION_BLOCK_CREATE, Disabled=FALSE)  // ARITH_0
        777 = ARITH_MODE+1 (Name=FUNCTION_BLOCK_CREATE, Disabled=FALSE)  // ARITH_1
        777 = ARITH_MODE+2 (Name=FUNCTION_BLOCK_CREATE, Disabled=FALSE)  // ARITH_2
        777 = ARITH_MODE+3 (Name=FUNCTION_BLOCK_CREATE, Disabled=FALSE)  // ARITH_3
        777 = ARITH_MODE+4 (Name=FUNCTION_BLOCK_CREATE, Disabled=FALSE)  // ARITH_4
        777 = ARITH_MODE+5 (Name=FUNCTION_BLOCK_CREATE, Disabled=FALSE)  // ARITH_5
        777 = MINMAX_MODE+0 (Name=FUNCTION_BLOCK_CREATE, Disabled=FALSE)  // MINMAX_0
        777 = MINMAX_MODE+1 (Name=FUNCTION_BLOCK_CREATE, Disabled=FALSE)  // MINMAX_1
        777 = EVWR_MODE+2 (Name=FUNCTION_BLOCK_CREATE, Disabled=FALSE)  // EVWR_2
        777 = EVWR_MODE+3 (Name=FUNCTION_BLOCK_CREATE, Disabled=FALSE)  // EVWR_3
        777 = EVWR_MODE+4 (Name=FUNCTION_BLOCK_CREATE, Disabled=FALSE)  // EVWR_4
        777 = EVWR_MODE+5 (Name=FUNCTION_BLOCK_CREATE, Disabled=FALSE)  // EVWR_5
      IPL (Disabled=FALSE)
        8713 = VAR_R4_1+0 (Name=IPL_IN_PARID+1, Disabled=FALSE)  // 4136
        8761 = CYCLIC_TODRV_COUNT (Name=IPL_EV_PARID+1, Disabled=FALSE)  // 909 - CYCLIC_TODRV_COUNT
        8721 = 2000 (Name=IPL_CYCLE_TIME+1, Unit=us, Disabled=FALSE)  // FB1 FB IPL: Cycle time
        8729 = 2000 (Name=IPL_EXTRAPOLATION_TIME+1, Unit=us, Disabled=FALSE)  // FB1 FB IPL: Extrapolation time
        8705 = 1 (Name=IPL_MODE+1, Disabled=FALSE)  // FB1 FB IPL: Mode -- linear interpolation
      ARITH + 0 (Disabled=FALSE)
        3592 = TEMP_JUNCTION_LIM (Name=ARITH_IN1_PARID+0, Disabled=FALSE)  // TEMP_JUNCTION_LIM -- 842
        3600 = TEMP_JUNCTION (Name=ARITH_IN2_PARID+0, Disabled=FALSE)  // TEMP_JUNCTION -- 382
        3632 = 0 (Name=ARITH_K1+0, Disabled=FALSE)  // FB0 FB ARITH: Multiplication factor1
        3640 = 0 (Name=ARITH_K2+0, Disabled=FALSE)  // FB0 FB ARITH: Multiplication factor2
        3584 = 2 (Name=ARITH_MODE+0, Disabled=FALSE)  // y= x1 - x2
      ARITH + 1 (Disabled=FALSE)
        3593 = ARITH_VALUE_R4+0 (Name=ARITH_IN1_PARID+1, Disabled=FALSE)  // 3624
        3601 = VAR_R4_2+0 (Name=ARITH_IN2_PARID+1, Disabled=FALSE)  // 4144
        3633 = 0 (Name=ARITH_K1+1, Disabled=FALSE)  // FB1 FB ARITH: Multiplication factor1
        3641 = 0 (Name=ARITH_K2+1, Disabled=FALSE)  // FB1 FB ARITH: Multiplication factor2
        3585 = 3 (Name=ARITH_MODE+1, Disabled=FALSE)  // y = x1 * x2
      ARITH + 2 (Disabled=FALSE)
        3594 = MOTOR_TORQ_RATED (Name=ARITH_IN1_PARID+2, Disabled=FALSE)  // MOTOR_TORQ_RATED -- 53
        3602 = ARITH_VALUE_R4+1 (Name=ARITH_IN2_PARID+2, Disabled=FALSE)  // 3625
        3634 = 0 (Name=ARITH_K1+2, Disabled=FALSE)  // FB2 FB ARITH: Multiplication factor1
        3642 = 0 (Name=ARITH_K2+2, Disabled=FALSE)  // FB2 FB ARITH: Multiplication factor2
        3586 = 1 (Name=ARITH_MODE+2, Disabled=FALSE)  // y = x1 + x2
      ARITH + 3 (Disabled=FALSE)
        3595 = MOTOR_WIND_TEMP_MAX (Name=ARITH_IN1_PARID+3, Disabled=FALSE)  // 74 - MOTOR_WIND_TEMP_MAX
        3603 = TEMP_MOTOR_MODELL (Name=ARITH_IN2_PARID+3, Disabled=FALSE)  // 393 - TEMP_MOTOR_MODELL   381 - TEMP_MOTOR
        3635 = 0 (Name=ARITH_K1+3, Disabled=FALSE)  // FB3 FB ARITH: Multiplication factor1
        3643 = 0 (Name=ARITH_K2+3, Disabled=FALSE)  // FB3 FB ARITH: Multiplication factor2
        3587 = 2 (Name=ARITH_MODE+3, Disabled=FALSE)  // y = x1 - x2
      ARITH + 4 (Disabled=FALSE)
        3596 = ARITH_VALUE_R4+3 (Name=ARITH_IN1_PARID+4, Disabled=FALSE)  // 3627
        3604 = VAR_R4_3+0 (Name=ARITH_IN2_PARID+4, Disabled=FALSE)  // 4152
        3636 = 0 (Name=ARITH_K1+4, Disabled=FALSE)  // FB4 FB ARITH: Multiplication factor1
        3644 = 0 (Name=ARITH_K2+4, Disabled=FALSE)  // FB4 FB ARITH: Multiplication factor2
        3588 = 3 (Name=ARITH_MODE+4, Disabled=FALSE)  // y = x1 * x2
      ARITH + 5 (Disabled=FALSE)
        3597 = MOTOR_TORQ_RATED (Name=ARITH_IN1_PARID+5, Disabled=FALSE)  // MOTOR_TORQ_RATED -- 53
        3605 = ARITH_VALUE_R4+4 (Name=ARITH_IN2_PARID+5, Disabled=FALSE)  // 3628
        3637 = 0 (Name=ARITH_K1+5, Disabled=FALSE)  // FB5 FB ARITH: Multiplication factor1
        3645 = 0 (Name=ARITH_K2+5, Disabled=FALSE)  // FB5 FB ARITH: Multiplication factor2
        3589 = 1 (Name=ARITH_MODE+5, Disabled=FALSE)  // y = x1 + x2
      MINMAX + 0 (Disabled=FALSE)
        12312 = VAR_R4_2+1 (Name=MINMAX_IN1_PARID+0, Disabled=FALSE)  // MOTOR_TORQ_MAX -- 54 / Torque_Max - User Setting
        12320 = ARITH_VALUE_R4+2 (Name=MINMAX_IN2_PARID+0, Disabled=FALSE)  // 3626
        12328 = ARITH_VALUE_R4+5 (Name=MINMAX_IN3_PARID+0, Disabled=FALSE)  // 3629
        12336 = IPL_VALUE_R4+1 (Name=MINMAX_IN4_PARID+0, Disabled=FALSE)  // 8753 -- interpolated torque set
        12288 = 1 (Name=MINMAX_MODE+0, Disabled=FALSE)  // MIN(MOTOR_TORQ_MAX,ARITH_VALUE_R4+1)
      MINMAX + 1 (Disabled=FALSE)
        12313 = VAR_R4_0+1 (Name=MINMAX_IN1_PARID+1, Disabled=FALSE)  // zero
        12321 = MINMAX_VALUE_R4+0 (Name=MINMAX_IN2_PARID+1, Disabled=FALSE)  // FB1 FB MINMAX: Parameter ID of input2
        12289 = 2 (Name=MINMAX_MODE+1, Disabled=FALSE)  // MAX(VAR_R4_0+1,MINMAX_VALUE_R4+0)
      EVWR + 2 (Disabled=FALSE)
        4610 = CONST_I4_ONE (Name=EVWR_EVENT_PARID+2, Disabled=FALSE)  // FB2 FB EVWR: Parameter ID of event input
        4618 = MINMAX_VALUE_R4+1 (Name=EVWR_IN_PARID+2, Disabled=FALSE)  // FB2 FB EVWR: Parameter ID of input
        4626 = 1 (Name=EVWR_EVENT_LEVEL+2, Disabled=FALSE)  // FB2 FB EVWR: Event level
        4634 = LIM_T2_POS (Name=EVWR_WR_PARID+2, Disabled=FALSE)  // 348
        4642 = 2 (Name=EVWR_MODE+2, Disabled=FALSE)  // mode - cyclic write
      EVWR + 3 (Disabled=FALSE)
        4611 = CONST_I4_ONE (Name=EVWR_EVENT_PARID+3, Disabled=FALSE)  // FB3 FB EVWR: Parameter ID of event input
        4619 = MINMAX_VALUE_R4+1 (Name=EVWR_IN_PARID+3, Disabled=FALSE)  // FB3 FB EVWR: Parameter ID of input
        4627 = 1 (Name=EVWR_EVENT_LEVEL+3, Disabled=FALSE)  // FB3 FB EVWR: Event level
        4635 = LIM_T2_NEG (Name=EVWR_WR_PARID+3, Disabled=FALSE)  // 349
        4643 = 2 (Name=EVWR_MODE+3, Disabled=FALSE)  // mode - cyclic write
      EVWR + 4 (Disabled=FALSE)
        4612 = CONST_I4_ONE (Name=EVWR_EVENT_PARID+4, Disabled=FALSE)  // FB4 FB EVWR: Parameter ID of event input
        4620 = MINMAX_VALUE_R4+1 (Name=EVWR_IN_PARID+4, Disabled=FALSE)  // FB4 FB EVWR: Parameter ID of input
        4628 = 1 (Name=EVWR_EVENT_LEVEL+4, Disabled=FALSE)  // FB4 FB EVWR: Event level
        4636 = LIM_T1_POS (Name=EVWR_WR_PARID+4, Disabled=FALSE)  // 248
        4644 = 2 (Name=EVWR_MODE+4, Disabled=FALSE)  // mode - cyclic write
      EVWR + 5 (Disabled=FALSE)
        4613 = CONST_I4_ONE (Name=EVWR_EVENT_PARID+5, Disabled=FALSE)  // FB5 FB EVWR: Parameter ID of event input
        4621 = MINMAX_VALUE_R4+1 (Name=EVWR_IN_PARID+5, Disabled=FALSE)  // FB5 FB EVWR: Parameter ID of input
        4629 = 1 (Name=EVWR_EVENT_LEVEL+5, Disabled=FALSE)  // FB5 FB EVWR: Event level
        4637 = LIM_T1_NEG (Name=EVWR_WR_PARID+5, Disabled=FALSE)  // 249
        4645 = 2 (Name=EVWR_MODE+5, Disabled=FALSE)  // mode - cyclic write
    HardWare Limit  For ACOPOS Multi (Disabled=FALSE)
      945 = VAR_I2_0+0 (Name=POS_LIMIT_SWITCH_PARID, Disabled=FALSE)  // Digital inputs: Parameter ID for positive end switch
      946 = VAR_I2_1+0 (Name=NEG_LIMIT_SWITCH_PARID, Disabled=FALSE)  // Digital inputs: Parameter ID for negative end switch
    90 = 0 (Name=BRAKE_MODE, Disabled=TRUE)  // Motor holding brake: Mode
```

### Data object Logical/Motion/para/ThickPara (Apt)

#### ThickPara.apt
```
AcoposParameterTable:
  Root Parameters:
    Configure Parameter (Disabled=FALSE)
      128 = 1 (Name=SGEN_SW_END_IGNORE, Disabled=FALSE)  // Limit values: Ignore SW end positions
      1196 = 0 (Name=PCTRL_MODE_BITS, Disabled=FALSE)  // CTRL Position controller: Mode bits
      90 = 0 (Name=BRAKE_MODE, Disabled=TRUE)  // Motor holding brake: Mode
      80 = 1 (Name=PHASE_MON_IGNORE, Disabled=FALSE)  // Power mains: Ignore phase failure
      300 = 300 (Name=UDC_DETECTION, Unit=V, Disabled=FALSE)  // CTRL DC bus: Voltage detection: Lower limit
    VAR_XX_X+0 (Disabled=FALSE)
      777 = VAR_I4_0+0 (Name=FUNCTION_BLOCK_CREATE, Disabled=FALSE)  // VAR_XX_X+0
      VAR_R4_X_0 (Disabled=FALSE)
        4128 = 0.0 (Name=VAR_R4_0+0, Disabled=FALSE)  // velocity set -- cyclic set
        4136 = 0.0 (Name=VAR_R4_1+0, Disabled=FALSE)  // torque limit -- cyclic set
        4144 = 0.97 (Name=VAR_R4_2+0, Disabled=FALSE)  // temp junction Kp
        4152 = 0.97 (Name=VAR_R4_3+0, Disabled=FALSE)  // temp motor Kp
    VAR_XX_X+1 (Disabled=FALSE)
      777 = VAR_I4_0+1 (Name=FUNCTION_BLOCK_CREATE, Disabled=FALSE)  // VAR_XX_X+1
      VAR_R4_X_1 (Disabled=FALSE)
        4129 = 0.0 (Name=VAR_R4_0+1, Disabled=FALSE)  // zero
        4137 = 0.0 (Name=VAR_R4_1+1, Disabled=FALSE)  // 288 - SCTRL_ADD_SET_PARID
        4145 = 12.6 (Name=VAR_R4_2+1, Disabled=FALSE)  // Torque_Max - User Setting
        4153 = 0.0 (Name=VAR_R4_3+1, Disabled=FALSE)  // no use
    VAR_XX_X+2 (Disabled=FALSE)
      777 = VAR_I4_0+2 (Name=FUNCTION_BLOCK_CREATE, Disabled=FALSE)  // VAR_XX_X+2
      VAR_R4_X_2 (Disabled=FALSE)
        4130 = 0.0 (Name=VAR_R4_0+2, Disabled=FALSE)  // Power Consumption Trigger - Left Carriage
        4138 = 0.0 (Name=VAR_R4_1+2, Disabled=FALSE)  // Power Consumption Trigger - Right Carriage
        4146 = 0.0 (Name=VAR_R4_2+2, Disabled=FALSE)  // FB2 FB VAR: Variable2 R4
        4154 = 0.0 (Name=VAR_R4_3+2, Disabled=FALSE)  // FB2 FB VAR: Variable3 R4
    Velocity Control (Disabled=FALSE)
      Function Create (Disabled=FALSE)
        777 = IPL_MODE+0 (Name=FUNCTION_BLOCK_CREATE, Disabled=FALSE)  // IPL_0
        777 = EVWR_MODE+0 (Name=FUNCTION_BLOCK_CREATE, Disabled=FALSE)  // EVWR_0
        777 = CMP_MODE+0 (Name=FUNCTION_BLOCK_CREATE, Disabled=FALSE)  // CMP_0
        777 = EVWR_MODE+1 (Name=FUNCTION_BLOCK_CREATE, Disabled=FALSE)  // EVWR_1
      IPL + 0 (Disabled=FALSE)
        8712 = VAR_R4_0+0 (Name=IPL_IN_PARID+0, Disabled=FALSE)  // velocity set
        8760 = CYCLIC_TODRV_COUNT (Name=IPL_EV_PARID+0, Disabled=FALSE)  // 909 - CYCLIC_TODRV_COUNT
        8720 = 2000 (Name=IPL_CYCLE_TIME+0, Unit=us, Disabled=FALSE)  // FB0 FB IPL: Cycle time
        8728 = 800 (Name=IPL_EXTRAPOLATION_TIME+0, Unit=us, Disabled=FALSE)  // FB0 FB IPL: Extrapolation time
        8704 = 1 (Name=IPL_MODE+0, Disabled=FALSE)  // linear interpolation
      EVWR + 0 (Disabled=FALSE)
        4608 = CMP_VALUE+0 (Name=EVWR_EVENT_PARID+0, Disabled=FALSE)  // v_set == 0
        4616 = IPL_VALUE_R4+0 (Name=EVWR_IN_PARID+0, Disabled=FALSE)  // 8752 -- interpolated v_set
        4624 = 0 (Name=EVWR_EVENT_LEVEL+0, Disabled=FALSE)  // FB0 FB EVWR: Event level
        4632 = VAR_R4_1+1 (Name=EVWR_WR_PARID+0, Disabled=FALSE)  // 288 - SCTRL_ADD_SET_PARID
        4640 = 2 (Name=EVWR_MODE+0, Disabled=FALSE)  // cyclic write
      288 = VAR_R4_1+1 (Name=SCTRL_ADD_SET_PARID, Disabled=FALSE)  // CTRL Speed controller: Parameter ID additive set value
      CMP + 0 (Disabled=FALSE)
        6656 = IPL_VALUE_R4+0 (Name=CMP_IN_PARID+0, Disabled=FALSE)  // 8752 -- interpolated v_set
        6664 = 0 (Name=CMP_THRESHOLD+0, Disabled=FALSE)  // FB0 FB CMP: threshold
        6672 = 0.001 (Name=CMP_WINDOW+0, Disabled=FALSE)  // FB0 FB CMP: window
        6680 = 0 (Name=CMP_HYSTERESIS+0, Disabled=FALSE)  // FB0 FB CMP: hysteresis window
        6688 = 2 (Name=CMP_MODE+0, Disabled=FALSE)  // ==
      231 = CMP_VALUE+0 (Name=PCTRL_ENABLE_PARID, Disabled=FALSE)  // if(interpolated v_set == 0)enable PCTRL
      EVWR + 1 (Disabled=FALSE)
        4609 = CMP_VALUE+0 (Name=EVWR_EVENT_PARID+1, Disabled=FALSE)  // 6696
        4617 = VAR_R4_2+1 (Name=EVWR_IN_PARID+1, Disabled=FALSE)  // FB1 FB EVWR: Parameter ID of input / Torque_Max - User Setting
        4625 = 1 (Name=EVWR_EVENT_LEVEL+1, Disabled=FALSE)  // FB1 FB EVWR: Event level
        4633 = VAR_R4_1+0 (Name=EVWR_WR_PARID+1, Disabled=FALSE)  // FB1 FB EVWR: Parameter ID of output value
        4641 = 2 (Name=EVWR_MODE+1, Disabled=FALSE)  // mode - cyclic write
    Torque Limitation (Disabled=FALSE)
      Function Create (Disabled=FALSE)
        777 = IPL_MODE+1 (Name=FUNCTION_BLOCK_CREATE, Disabled=FALSE)  // IPL_1
        777 = ARITH_MODE+0 (Name=FUNCTION_BLOCK_CREATE, Disabled=FALSE)  // ARITH_0
        777 = ARITH_MODE+1 (Name=FUNCTION_BLOCK_CREATE, Disabled=FALSE)  // ARITH_1
        777 = ARITH_MODE+2 (Name=FUNCTION_BLOCK_CREATE, Disabled=FALSE)  // ARITH_2
        777 = ARITH_MODE+3 (Name=FUNCTION_BLOCK_CREATE, Disabled=FALSE)  // ARITH_3
        777 = ARITH_MODE+4 (Name=FUNCTION_BLOCK_CREATE, Disabled=FALSE)  // ARITH_4
        777 = ARITH_MODE+5 (Name=FUNCTION_BLOCK_CREATE, Disabled=FALSE)  // ARITH_5
        777 = MINMAX_MODE+0 (Name=FUNCTION_BLOCK_CREATE, Disabled=FALSE)  // MINMAX_0
        777 = MINMAX_MODE+1 (Name=FUNCTION_BLOCK_CREATE, Disabled=FALSE)  // MINMAX_1
        777 = EVWR_MODE+2 (Name=FUNCTION_BLOCK_CREATE, Disabled=FALSE)  // EVWR_2
        777 = EVWR_MODE+3 (Name=FUNCTION_BLOCK_CREATE, Disabled=FALSE)  // EVWR_3
        777 = EVWR_MODE+4 (Name=FUNCTION_BLOCK_CREATE, Disabled=FALSE)  // EVWR_4
        777 = EVWR_MODE+5 (Name=FUNCTION_BLOCK_CREATE, Disabled=FALSE)  // EVWR_5
      IPL (Disabled=FALSE)
        8713 = VAR_R4_1+0 (Name=IPL_IN_PARID+1, Disabled=FALSE)  // 4136
        8761 = CYCLIC_TODRV_COUNT (Name=IPL_EV_PARID+1, Disabled=FALSE)  // 909 - CYCLIC_TODRV_COUNT
        8721 = 2000 (Name=IPL_CYCLE_TIME+1, Unit=us, Disabled=FALSE)  // FB1 FB IPL: Cycle time
        8729 = 2000 (Name=IPL_EXTRAPOLATION_TIME+1, Unit=us, Disabled=FALSE)  // FB1 FB IPL: Extrapolation time
        8705 = 1 (Name=IPL_MODE+1, Disabled=FALSE)  // FB1 FB IPL: Mode -- linear interpolation
      ARITH + 0 (Disabled=FALSE)
        3592 = TEMP_JUNCTION_LIM (Name=ARITH_IN1_PARID+0, Disabled=FALSE)  // TEMP_JUNCTION_LIM -- 842
        3600 = TEMP_JUNCTION (Name=ARITH_IN2_PARID+0, Disabled=FALSE)  // TEMP_JUNCTION -- 382
        3632 = 0 (Name=ARITH_K1+0, Disabled=FALSE)  // FB0 FB ARITH: Multiplication factor1
        3640 = 0 (Name=ARITH_K2+0, Disabled=FALSE)  // FB0 FB ARITH: Multiplication factor2
        3584 = 2 (Name=ARITH_MODE+0, Disabled=FALSE)  // y= x1 - x2
      ARITH + 1 (Disabled=FALSE)
        3593 = ARITH_VALUE_R4+0 (Name=ARITH_IN1_PARID+1, Disabled=FALSE)  // 3624
        3601 = VAR_R4_2+0 (Name=ARITH_IN2_PARID+1, Disabled=FALSE)  // 4144
        3633 = 0 (Name=ARITH_K1+1, Disabled=FALSE)  // FB1 FB ARITH: Multiplication factor1
        3641 = 0 (Name=ARITH_K2+1, Disabled=FALSE)  // FB1 FB ARITH: Multiplication factor2
        3585 = 3 (Name=ARITH_MODE+1, Disabled=FALSE)  // y = x1 * x2
      ARITH + 2 (Disabled=FALSE)
        3594 = MOTOR_TORQ_RATED (Name=ARITH_IN1_PARID+2, Disabled=FALSE)  // MOTOR_TORQ_RATED -- 53
        3602 = ARITH_VALUE_R4+1 (Name=ARITH_IN2_PARID+2, Disabled=FALSE)  // 3625
        3634 = 0 (Name=ARITH_K1+2, Disabled=FALSE)  // FB2 FB ARITH: Multiplication factor1
        3642 = 0 (Name=ARITH_K2+2, Disabled=FALSE)  // FB2 FB ARITH: Multiplication factor2
        3586 = 1 (Name=ARITH_MODE+2, Disabled=FALSE)  // y = x1 + x2
      ARITH + 3 (Disabled=FALSE)
        3595 = MOTOR_WIND_TEMP_MAX (Name=ARITH_IN1_PARID+3, Disabled=FALSE)  // 74 - MOTOR_WIND_TEMP_MAX
        3603 = TEMP_MOTOR_MODELL (Name=ARITH_IN2_PARID+3, Disabled=FALSE)  // 393 - TEMP_MOTOR_MODELL
        3635 = 0 (Name=ARITH_K1+3, Disabled=FALSE)  // FB3 FB ARITH: Multiplication factor1
        3643 = 0 (Name=ARITH_K2+3, Disabled=FALSE)  // FB3 FB ARITH: Multiplication factor2
        3587 = 2 (Name=ARITH_MODE+3, Disabled=FALSE)  // y = x1 - x2
      ARITH + 4 (Disabled=FALSE)
        3596 = ARITH_VALUE_R4+3 (Name=ARITH_IN1_PARID+4, Disabled=FALSE)  // 3627
        3604 = VAR_R4_3+0 (Name=ARITH_IN2_PARID+4, Disabled=FALSE)  // 4152
        3636 = 0 (Name=ARITH_K1+4, Disabled=FALSE)  // FB4 FB ARITH: Multiplication factor1
        3644 = 0 (Name=ARITH_K2+4, Disabled=FALSE)  // FB4 FB ARITH: Multiplication factor2
        3588 = 3 (Name=ARITH_MODE+4, Disabled=FALSE)  // y = x1 * x2
      ARITH + 5 (Disabled=FALSE)
        3597 = MOTOR_TORQ_RATED (Name=ARITH_IN1_PARID+5, Disabled=FALSE)  // MOTOR_TORQ_RATED -- 53
        3605 = ARITH_VALUE_R4+4 (Name=ARITH_IN2_PARID+5, Disabled=FALSE)  // 3628
        3637 = 0 (Name=ARITH_K1+5, Disabled=FALSE)  // FB5 FB ARITH: Multiplication factor1
        3645 = 0 (Name=ARITH_K2+5, Disabled=FALSE)  // FB5 FB ARITH: Multiplication factor2
        3589 = 1 (Name=ARITH_MODE+5, Disabled=FALSE)  // y = x1 + x2
      MINMAX + 0 (Disabled=FALSE)
        12312 = VAR_R4_2+1 (Name=MINMAX_IN1_PARID+0, Disabled=FALSE)  // MOTOR_TORQ_MAX -- 54 / Torque_Max - User Setting
        12320 = ARITH_VALUE_R4+2 (Name=MINMAX_IN2_PARID+0, Disabled=FALSE)  // 3626
        12328 = ARITH_VALUE_R4+5 (Name=MINMAX_IN3_PARID+0, Disabled=FALSE)  // 3629
        12336 = IPL_VALUE_R4+1 (Name=MINMAX_IN4_PARID+0, Disabled=FALSE)  // 8753 -- interpolated torque set
        12288 = 1 (Name=MINMAX_MODE+0, Disabled=FALSE)  // MIN(MOTOR_TORQ_MAX,ARITH_VALUE_R4+1)
      MINMAX + 1 (Disabled=FALSE)
        12313 = VAR_R4_0+1 (Name=MINMAX_IN1_PARID+1, Disabled=FALSE)  // zero
        12321 = MINMAX_VALUE_R4+0 (Name=MINMAX_IN2_PARID+1, Disabled=FALSE)  // FB1 FB MINMAX: Parameter ID of input2
        12289 = 2 (Name=MINMAX_MODE+1, Disabled=FALSE)  // MAX(VAR_R4_0+1,MINMAX_VALUE_R4+0)
      EVWR + 2 (Disabled=FALSE)
        4610 = CONST_I4_ONE (Name=EVWR_EVENT_PARID+2, Disabled=FALSE)  // FB2 FB EVWR: Parameter ID of event input
        4618 = MINMAX_VALUE_R4+1 (Name=EVWR_IN_PARID+2, Disabled=FALSE)  // FB2 FB EVWR: Parameter ID of input
        4626 = 1 (Name=EVWR_EVENT_LEVEL+2, Disabled=FALSE)  // FB2 FB EVWR: Event level
        4634 = LIM_T2_POS (Name=EVWR_WR_PARID+2, Disabled=FALSE)  // 348
        4642 = 2 (Name=EVWR_MODE+2, Disabled=FALSE)  // mode - cyclic write
      EVWR + 3 (Disabled=FALSE)
        4611 = CONST_I4_ONE (Name=EVWR_EVENT_PARID+3, Disabled=FALSE)  // FB3 FB EVWR: Parameter ID of event input
        4619 = MINMAX_VALUE_R4+1 (Name=EVWR_IN_PARID+3, Disabled=FALSE)  // FB3 FB EVWR: Parameter ID of input
        4627 = 1 (Name=EVWR_EVENT_LEVEL+3, Disabled=FALSE)  // FB3 FB EVWR: Event level
        4635 = LIM_T2_NEG (Name=EVWR_WR_PARID+3, Disabled=FALSE)  // 349
        4643 = 2 (Name=EVWR_MODE+3, Disabled=FALSE)  // mode - cyclic write
      EVWR + 4 (Disabled=FALSE)
        4612 = CONST_I4_ONE (Name=EVWR_EVENT_PARID+4, Disabled=FALSE)  // FB4 FB EVWR: Parameter ID of event input
        4620 = MINMAX_VALUE_R4+1 (Name=EVWR_IN_PARID+4, Disabled=FALSE)  // FB4 FB EVWR: Parameter ID of input
        4628 = 1 (Name=EVWR_EVENT_LEVEL+4, Disabled=FALSE)  // FB4 FB EVWR: Event level
        4636 = LIM_T1_POS (Name=EVWR_WR_PARID+4, Disabled=FALSE)  // 248
        4644 = 2 (Name=EVWR_MODE+4, Disabled=FALSE)  // mode - cyclic write
      EVWR + 5 (Disabled=FALSE)
        4613 = CONST_I4_ONE (Name=EVWR_EVENT_PARID+5, Disabled=FALSE)  // FB5 FB EVWR: Parameter ID of event input
        4621 = MINMAX_VALUE_R4+1 (Name=EVWR_IN_PARID+5, Disabled=FALSE)  // FB5 FB EVWR: Parameter ID of input
        4629 = 1 (Name=EVWR_EVENT_LEVEL+5, Disabled=FALSE)  // FB5 FB EVWR: Event level
        4637 = LIM_T1_NEG (Name=EVWR_WR_PARID+5, Disabled=FALSE)  // 249
        4645 = 2 (Name=EVWR_MODE+5, Disabled=FALSE)  // mode - cyclic write
    Position Control (Disabled=FALSE)
      777 = LOGIC_MODE+0 (Name=FUNCTION_BLOCK_CREATE, Disabled=FALSE)  // Function block: Create a FB instance
      777 = IPL_MODE+2 (Name=FUNCTION_BLOCK_CREATE, Disabled=FALSE)  // Function block: Create a FB instance
      777 = EVWR_MODE+6 (Name=FUNCTION_BLOCK_CREATE, Disabled=FALSE)  // Function block: Create a FB instance
      IPL (Disabled=FALSE)
        8714 = VAR_I4_0+0 (Name=IPL_IN_PARID+2, Disabled=FALSE)  // FB0 IPL Parameter ID of input
        8762 = CYCLIC_TODRV_COUNT (Name=IPL_EV_PARID+2, Disabled=FALSE)  // FB0 IPL Parameter ID of event input
        8722 = 2000 (Name=IPL_CYCLE_TIME+2, Unit=us, Disabled=FALSE)  // FB0 IPL Cycle time
        8730 = 800 (Name=IPL_EXTRAPOLATION_TIME+2, Unit=us, Disabled=FALSE)  // FB0 IPL Extrapolation time
        8706 = 1 (Name=IPL_MODE+2, Disabled=FALSE)  // FB0 IPL Mode
      LOGIC (Disabled=FALSE)
        3080 = VAR_UI1_0+0 (Name=LOGIC_IN1_PARID+0, Disabled=FALSE)  // FB0 LOGIC Parameter ID of input1 --- auto run thick
        3088 = CMP_VALUE+0 (Name=LOGIC_IN2_PARID+0, Disabled=FALSE)  // FB0 LOGIC Parameter ID of input2  --- position loop
        3072 = 8 (Name=LOGIC_MODE+0, Disabled=FALSE)  // FB0 LOGIC Mode    ---- and
      EVWR (Disabled=FALSE)
        4614 = LOGIC_VALUE+0 (Name=EVWR_EVENT_PARID+6, Disabled=FALSE)  // Thick auto run and position mode
        4622 = IPL_VALUE_I4+2 (Name=EVWR_IN_PARID+6, Disabled=FALSE)  // IPL set position
        4630 = 1 (Name=EVWR_EVENT_LEVEL+6, Disabled=FALSE)  // FB0 EVWR Event level
        4638 = CMD_ABS_MOVE (Name=EVWR_WR_PARID+6, Disabled=FALSE)  // abs move position and command
        4646 = 2 (Name=EVWR_MODE+6, Disabled=FALSE)  // CYCLIC WRITE
```

### Data object Logical/Motion/para/ExtrLift (Apt)

#### ExtrLift.apt
```
AcoposParameterTable:
  Root Parameters:
    Configure Parameter (Disabled=FALSE)
      128 = 1 (Name=SGEN_SW_END_IGNORE, Disabled=FALSE)  // Limit values: Ignore SW end positions
      1196 = 0 (Name=PCTRL_MODE_BITS, Disabled=FALSE)  // CTRL Position controller: Mode bits
      80 = 1 (Name=PHASE_MON_IGNORE, Disabled=FALSE)  // Power mains: Ignore phase failure
      300 = 300 (Name=UDC_DETECTION, Unit=V)  // CTRL DC bus: Voltage detection: Lower limit
    VAR_XX_X+0 (Disabled=FALSE)
      777 = VAR_I4_0+0 (Name=FUNCTION_BLOCK_CREATE, Disabled=FALSE)  // VAR_XX_X+0
      VAR_R4_X_0 (Disabled=FALSE)
        4128 = 0.0 (Name=VAR_R4_0+0, Disabled=FALSE)  // velocity set -- cyclic set
        4136 = 0.0 (Name=VAR_R4_1+0, Disabled=FALSE)  // torque limit -- cyclic set
        4144 = 0.363 (Name=VAR_R4_2+0, Disabled=FALSE)  // temp junction Kp
        4152 = 0.363 (Name=VAR_R4_3+0, Disabled=FALSE)  // temp motor Kp
    VAR_XX_X+1 (Disabled=FALSE)
      777 = VAR_I4_0+1 (Name=FUNCTION_BLOCK_CREATE, Disabled=FALSE)  // VAR_XX_X+1
      VAR_R4_X_1 (Disabled=FALSE)
        4129 = 0.0 (Name=VAR_R4_0+1, Disabled=FALSE)  // zero
        4137 = 0.0 (Name=VAR_R4_1+1, Disabled=FALSE)  // 288 - SCTRL_ADD_SET_PARID
        4145 = 3.3 (Name=VAR_R4_2+1, Disabled=FALSE)  // Torque_Max - User Setting
        4153 = 0.0 (Name=VAR_R4_3+1, Disabled=FALSE)  // no use
      VAR_XX_X+2 (Disabled=FALSE)
        777 = VAR_I4_0+2 (Name=FUNCTION_BLOCK_CREATE, Disabled=FALSE)  // VAR_XX_X+2
        VAR_R4_X_2 (Disabled=FALSE)
          4130 = 0.0 (Name=VAR_R4_0+2, Disabled=FALSE)  // Power Consumption Trigger - Left Carriage
          4138 = 0.0 (Name=VAR_R4_1+2, Disabled=FALSE)  // Power Consumption Trigger - Right Carriage
          4146 = 0.0 (Name=VAR_R4_2+2, Disabled=FALSE)  // FB2 FB VAR: Variable2 R4
          4154 = 0.0 (Name=VAR_R4_3+2, Disabled=FALSE)  // FB2 FB VAR: Variable3 R4
    Velocity Control (Disabled=FALSE)
      Function Create (Disabled=FALSE)
        777 = IPL_MODE+0 (Name=FUNCTION_BLOCK_CREATE, Disabled=FALSE)  // IPL_0
        777 = EVWR_MODE+0 (Name=FUNCTION_BLOCK_CREATE, Disabled=FALSE)  // EVWR_0
        777 = CMP_MODE+0 (Name=FUNCTION_BLOCK_CREATE, Disabled=FALSE)  // CMP_0
        777 = EVWR_MODE+1 (Name=FUNCTION_BLOCK_CREATE, Disabled=FALSE)  // EVWR_1
      IPL + 0 (Disabled=FALSE)
        8712 = VAR_R4_0+0 (Name=IPL_IN_PARID+0, Disabled=FALSE)  // velocity set
        8760 = CYCLIC_TODRV_COUNT (Name=IPL_EV_PARID+0, Disabled=FALSE)  // 909 - CYCLIC_TODRV_COUNT
        8720 = 2000 (Name=IPL_CYCLE_TIME+0, Unit=us, Disabled=FALSE)  // FB0 FB IPL: Cycle time
        8728 = 800 (Name=IPL_EXTRAPOLATION_TIME+0, Unit=us, Disabled=FALSE)  // FB0 FB IPL: Extrapolation time
        8704 = 1 (Name=IPL_MODE+0, Disabled=FALSE)  // linear interpolation
      EVWR + 0 (Disabled=FALSE)
        4608 = CMP_VALUE+0 (Name=EVWR_EVENT_PARID+0, Disabled=FALSE)  // v_set == 0
        4616 = IPL_VALUE_R4+0 (Name=EVWR_IN_PARID+0, Disabled=FALSE)  // 8752 -- interpolated v_set
        4624 = 0 (Name=EVWR_EVENT_LEVEL+0, Disabled=FALSE)  // FB0 FB EVWR: Event level
        4632 = VAR_R4_1+1 (Name=EVWR_WR_PARID+0, Disabled=FALSE)  // 288 - SCTRL_ADD_SET_PARID
        4640 = 2 (Name=EVWR_MODE+0, Disabled=FALSE)  // cyclic write
      288 = VAR_R4_1+1 (Name=SCTRL_ADD_SET_PARID, Disabled=FALSE)  // CTRL Speed controller: Parameter ID additive set value
      CMP + 0 (Disabled=FALSE)
        6656 = IPL_VALUE_R4+0 (Name=CMP_IN_PARID+0, Disabled=FALSE)  // 8752 -- interpolated v_set
        6664 = 0 (Name=CMP_THRESHOLD+0, Disabled=FALSE)  // FB0 FB CMP: threshold
        6672 = 0.001 (Name=CMP_WINDOW+0, Disabled=FALSE)  // FB0 FB CMP: window
        6680 = 0 (Name=CMP_HYSTERESIS+0, Disabled=FALSE)  // FB0 FB CMP: hysteresis window
        6688 = 2 (Name=CMP_MODE+0, Disabled=FALSE)  // ==
      231 = CMP_VALUE+0 (Name=PCTRL_ENABLE_PARID, Disabled=FALSE)  // if(interpolated v_set == 0)enable PCTRL
      EVWR + 1 (Disabled=FALSE)
        4609 = CMP_VALUE+0 (Name=EVWR_EVENT_PARID+1, Disabled=FALSE)  // 6696
        4617 = VAR_R4_2+1 (Name=EVWR_IN_PARID+1, Disabled=FALSE)  // FB1 FB EVWR: Parameter ID of input / Torque_Max - User Setting
        4625 = 1 (Name=EVWR_EVENT_LEVEL+1, Disabled=FALSE)  // FB1 FB EVWR: Event level
        4633 = VAR_R4_1+0 (Name=EVWR_WR_PARID+1, Disabled=FALSE)  // FB1 FB EVWR: Parameter ID of output value
        4641 = 2 (Name=EVWR_MODE+1, Disabled=FALSE)  // mode - cyclic write
    Torque Limitation (Disabled=FALSE)
      Function Create (Disabled=FALSE)
        777 = IPL_MODE+1 (Name=FUNCTION_BLOCK_CREATE, Disabled=FALSE)  // IPL_1
        777 = ARITH_MODE+0 (Name=FUNCTION_BLOCK_CREATE, Disabled=FALSE)  // ARITH_0
        777 = ARITH_MODE+1 (Name=FUNCTION_BLOCK_CREATE, Disabled=FALSE)  // ARITH_1
        777 = ARITH_MODE+2 (Name=FUNCTION_BLOCK_CREATE, Disabled=FALSE)  // ARITH_2
        777 = ARITH_MODE+3 (Name=FUNCTION_BLOCK_CREATE, Disabled=FALSE)  // ARITH_3
        777 = ARITH_MODE+4 (Name=FUNCTION_BLOCK_CREATE, Disabled=FALSE)  // ARITH_4
        777 = ARITH_MODE+5 (Name=FUNCTION_BLOCK_CREATE, Disabled=FALSE)  // ARITH_5
        777 = MINMAX_MODE+0 (Name=FUNCTION_BLOCK_CREATE, Disabled=FALSE)  // MINMAX_0
        777 = MINMAX_MODE+1 (Name=FUNCTION_BLOCK_CREATE, Disabled=FALSE)  // MINMAX_1
        777 = EVWR_MODE+2 (Name=FUNCTION_BLOCK_CREATE, Disabled=FALSE)  // EVWR_2
        777 = EVWR_MODE+3 (Name=FUNCTION_BLOCK_CREATE, Disabled=FALSE)  // EVWR_3
        777 = EVWR_MODE+4 (Name=FUNCTION_BLOCK_CREATE, Disabled=FALSE)  // EVWR_4
        777 = EVWR_MODE+5 (Name=FUNCTION_BLOCK_CREATE, Disabled=FALSE)  // EVWR_5
      IPL (Disabled=FALSE)
        8713 = VAR_R4_1+0 (Name=IPL_IN_PARID+1, Disabled=FALSE)  // 4136
        8761 = CYCLIC_TODRV_COUNT (Name=IPL_EV_PARID+1, Disabled=FALSE)  // 909 - CYCLIC_TODRV_COUNT
        8721 = 2000 (Name=IPL_CYCLE_TIME+1, Unit=us, Disabled=FALSE)  // FB1 FB IPL: Cycle time
        8729 = 2000 (Name=IPL_EXTRAPOLATION_TIME+1, Unit=us, Disabled=FALSE)  // FB1 FB IPL: Extrapolation time
        8705 = 1 (Name=IPL_MODE+1, Disabled=FALSE)  // FB1 FB IPL: Mode -- linear interpolation
      ARITH + 0 (Disabled=FALSE)
        3592 = TEMP_JUNCTION_LIM (Name=ARITH_IN1_PARID+0, Disabled=FALSE)  // TEMP_JUNCTION_LIM -- 842
        3600 = TEMP_JUNCTION (Name=ARITH_IN2_PARID+0, Disabled=FALSE)  // TEMP_JUNCTION -- 382
        3632 = 0 (Name=ARITH_K1+0, Disabled=FALSE)  // FB0 FB ARITH: Multiplication factor1
        3640 = 0 (Name=ARITH_K2+0, Disabled=FALSE)  // FB0 FB ARITH: Multiplication factor2
        3584 = 2 (Name=ARITH_MODE+0, Disabled=FALSE)  // y= x1 - x2
      ARITH + 1 (Disabled=FALSE)
        3593 = ARITH_VALUE_R4+0 (Name=ARITH_IN1_PARID+1, Disabled=FALSE)  // 3624
        3601 = VAR_R4_2+0 (Name=ARITH_IN2_PARID+1, Disabled=FALSE)  // 4144
        3633 = 0 (Name=ARITH_K1+1, Disabled=FALSE)  // FB1 FB ARITH: Multiplication factor1
        3641 = 0 (Name=ARITH_K2+1, Disabled=FALSE)  // FB1 FB ARITH: Multiplication factor2
        3585 = 3 (Name=ARITH_MODE+1, Disabled=FALSE)  // y = x1 * x2
      ARITH + 2 (Disabled=FALSE)
        3594 = MOTOR_TORQ_RATED (Name=ARITH_IN1_PARID+2, Disabled=FALSE)  // MOTOR_TORQ_RATED -- 53
        3602 = ARITH_VALUE_R4+1 (Name=ARITH_IN2_PARID+2, Disabled=FALSE)  // 3625
        3634 = 0 (Name=ARITH_K1+2, Disabled=FALSE)  // FB2 FB ARITH: Multiplication factor1
        3642 = 0 (Name=ARITH_K2+2, Disabled=FALSE)  // FB2 FB ARITH: Multiplication factor2
        3586 = 1 (Name=ARITH_MODE+2, Disabled=FALSE)  // y = x1 + x2
      ARITH + 3 (Disabled=FALSE)
        3595 = MOTOR_WIND_TEMP_MAX (Name=ARITH_IN1_PARID+3, Disabled=FALSE)  // 74 - MOTOR_WIND_TEMP_MAX
        3603 = TEMP_MOTOR_MODELL (Name=ARITH_IN2_PARID+3, Disabled=FALSE)  // 393 - TEMP_MOTOR_MODELL   381 - TEMP_MOTOR
        3635 = 0 (Name=ARITH_K1+3, Disabled=FALSE)  // FB3 FB ARITH: Multiplication factor1
        3643 = 0 (Name=ARITH_K2+3, Disabled=FALSE)  // FB3 FB ARITH: Multiplication factor2
        3587 = 2 (Name=ARITH_MODE+3, Disabled=FALSE)  // y = x1 - x2
      ARITH + 4 (Disabled=FALSE)
        3596 = ARITH_VALUE_R4+3 (Name=ARITH_IN1_PARID+4, Disabled=FALSE)  // 3627
        3604 = VAR_R4_3+0 (Name=ARITH_IN2_PARID+4, Disabled=FALSE)  // 4152
        3636 = 0 (Name=ARITH_K1+4, Disabled=FALSE)  // FB4 FB ARITH: Multiplication factor1
        3644 = 0 (Name=ARITH_K2+4, Disabled=FALSE)  // FB4 FB ARITH: Multiplication factor2
        3588 = 3 (Name=ARITH_MODE+4, Disabled=FALSE)  // y = x1 * x2
      ARITH + 5 (Disabled=FALSE)
        3597 = MOTOR_TORQ_RATED (Name=ARITH_IN1_PARID+5, Disabled=FALSE)  // MOTOR_TORQ_RATED -- 53
        3605 = ARITH_VALUE_R4+4 (Name=ARITH_IN2_PARID+5, Disabled=FALSE)  // 3628
        3637 = 0 (Name=ARITH_K1+5, Disabled=FALSE)  // FB5 FB ARITH: Multiplication factor1
        3645 = 0 (Name=ARITH_K2+5, Disabled=FALSE)  // FB5 FB ARITH: Multiplication factor2
        3589 = 1 (Name=ARITH_MODE+5, Disabled=FALSE)  // y = x1 + x2
      MINMAX + 0 (Disabled=FALSE)
        12312 = VAR_R4_2+1 (Name=MINMAX_IN1_PARID+0, Disabled=FALSE)  // MOTOR_TORQ_MAX -- 54 / Torque_Max - User Setting
        12320 = ARITH_VALUE_R4+2 (Name=MINMAX_IN2_PARID+0, Disabled=FALSE)  // 3626
        12328 = ARITH_VALUE_R4+5 (Name=MINMAX_IN3_PARID+0, Disabled=FALSE)  // 3629
        12336 = IPL_VALUE_R4+1 (Name=MINMAX_IN4_PARID+0, Disabled=FALSE)  // 8753 -- interpolated torque set
        12288 = 1 (Name=MINMAX_MODE+0, Disabled=FALSE)  // MIN(MOTOR_TORQ_MAX,ARITH_VALUE_R4+1)
      MINMAX + 1 (Disabled=FALSE)
        12313 = VAR_R4_0+1 (Name=MINMAX_IN1_PARID+1, Disabled=FALSE)  // zero
        12321 = MINMAX_VALUE_R4+0 (Name=MINMAX_IN2_PARID+1, Disabled=FALSE)  // FB1 FB MINMAX: Parameter ID of input2
        12289 = 2 (Name=MINMAX_MODE+1, Disabled=FALSE)  // MAX(VAR_R4_0+1,MINMAX_VALUE_R4+0)
      EVWR + 2 (Disabled=FALSE)
        4610 = CONST_I4_ONE (Name=EVWR_EVENT_PARID+2, Disabled=FALSE)  // FB2 FB EVWR: Parameter ID of event input
        4618 = MINMAX_VALUE_R4+1 (Name=EVWR_IN_PARID+2, Disabled=FALSE)  // FB2 FB EVWR: Parameter ID of input
        4626 = 1 (Name=EVWR_EVENT_LEVEL+2, Disabled=FALSE)  // FB2 FB EVWR: Event level
        4634 = LIM_T2_POS (Name=EVWR_WR_PARID+2, Disabled=FALSE)  // 348
        4642 = 2 (Name=EVWR_MODE+2, Disabled=FALSE)  // mode - cyclic write
      EVWR + 3 (Disabled=FALSE)
        4611 = CONST_I4_ONE (Name=EVWR_EVENT_PARID+3, Disabled=FALSE)  // FB3 FB EVWR: Parameter ID of event input
        4619 = MINMAX_VALUE_R4+1 (Name=EVWR_IN_PARID+3, Disabled=FALSE)  // FB3 FB EVWR: Parameter ID of input
        4627 = 1 (Name=EVWR_EVENT_LEVEL+3, Disabled=FALSE)  // FB3 FB EVWR: Event level
        4635 = LIM_T2_NEG (Name=EVWR_WR_PARID+3, Disabled=FALSE)  // 349
        4643 = 2 (Name=EVWR_MODE+3, Disabled=FALSE)  // mode - cyclic write
      EVWR + 4 (Disabled=FALSE)
        4612 = CONST_I4_ONE (Name=EVWR_EVENT_PARID+4, Disabled=FALSE)  // FB4 FB EVWR: Parameter ID of event input
        4620 = MINMAX_VALUE_R4+1 (Name=EVWR_IN_PARID+4, Disabled=FALSE)  // FB4 FB EVWR: Parameter ID of input
        4628 = 1 (Name=EVWR_EVENT_LEVEL+4, Disabled=FALSE)  // FB4 FB EVWR: Event level
        4636 = LIM_T1_POS (Name=EVWR_WR_PARID+4, Disabled=FALSE)  // 248
        4644 = 2 (Name=EVWR_MODE+4, Disabled=FALSE)  // mode - cyclic write
      EVWR + 5 (Disabled=FALSE)
        4613 = CONST_I4_ONE (Name=EVWR_EVENT_PARID+5, Disabled=FALSE)  // FB5 FB EVWR: Parameter ID of event input
        4621 = MINMAX_VALUE_R4+1 (Name=EVWR_IN_PARID+5, Disabled=FALSE)  // FB5 FB EVWR: Parameter ID of input
        4629 = 1 (Name=EVWR_EVENT_LEVEL+5, Disabled=FALSE)  // FB5 FB EVWR: Event level
        4637 = LIM_T1_NEG (Name=EVWR_WR_PARID+5, Disabled=FALSE)  // 249
        4645 = 2 (Name=EVWR_MODE+5, Disabled=FALSE)  // mode - cyclic write
    HardWare Limit  For ACOPOS Multi:
      945 = VAR_I2_0+0 (Name=POS_LIMIT_SWITCH_PARID)  // Digital inputs: Parameter ID for positive end switch
      946 = VAR_I2_1+0 (Name=NEG_LIMIT_SWITCH_PARID)  // Digital inputs: Parameter ID for negative end switch
```

### Program Logical/Motion/l_transfer (ANSIC) - left robot transfer

#### Types.typ
```iecst
TYPE
	Axis_ID_typ : 	STRUCT
		Address : UDINT; (*Address of the axis object data*)
		Name : STRING[20]; (*Logical name of the axis*)
		UnitFactor : REAL; (*Factor to calculate the displayed units*)
		UnitName : STRING[8]; (*Name of the unit to be displayed (e.g. deg,mm..)*)
		AxisType : UINT; (*ncAXIS or ncV_AXIS*)
	END_STRUCT;
	Axis_Status_typ : 	STRUCT
		ActPosition : REAL; (*actual position*)
		ActVelocity : REAL; (*actual velocity*)
		ActTorq : REAL; (*act torque*)
		ErrorID : UINT; (*Shows the Error ID (0 = No Error)*)
		ErrorText : ARRAY[0..3]OF STRING[79]; (*Shows the Acopos Errortext as string*)
	END_STRUCT;
	Axis_State_typ : 	STRUCT
		Disabled : BOOL; (*Status power disabled*)
		Standstill : BOOL; (*Status axis at standstill*)
		Stopping : BOOL; (*Status axis is stopping*)
		Homing : BOOL; (*Status axis is homing*)
		MotionDiscrete : BOOL; (*Status discrete motion is active*)
		MotionContinous : BOOL; (*Status continous motion is active*)
		MotionSynchronized : BOOL; (*Status synchronized motion is active*)
		ErrorStop : BOOL; (*Status axis stopped after error*)
	END_STRUCT;
	Axis_Parameter_typ : 	STRUCT
		Position : REAL; (*Parameter absolute target position*)
		Distance : REAL; (*Parameter relative move distance*)
		Velocity : REAL; (*Parameter target velocity*)
		Direction : USINT; (*Parameter movement direction*)
		Acceleration : REAL; (*Parameter movement acceleration*)
		Deceleration : REAL; (*Parameter movement deceleration*)
		HomePosition : REAL; (*Parameter home position*)
		HomeMode : USINT; (*Parameter homing mode*)
		JogVelocity : REAL; (*Parameter jog movement target velocity*)
		OverrideVelocity : REAL; (*Parameter velocity override (0.0 - 2.0)*)
		OverrideAcceleration : REAL; (*Parameter acceleration override (0.0001 - 2.0)*)
	END_STRUCT;
	Axis_Cmd_typ : 	STRUCT
		Init : BOOL; (*Download encoder parameter*)
		Power : BOOL; (*Turns the power on*)
		Home : BOOL; (*homes the axis*)
		MoveAbsolute : BOOL; (*Starts the absolute movement*)
		MoveAdditive : BOOL; (*Starts the additive movement*)
		MoveVelocity : BOOL; (*Starts the velocity movement*)
		Halt : BOOL; (*Stop every active movement*)
		Stop : BOOL; (*Stop every active movement as long as is set*)
		MoveJogPos : BOOL; (*Starts the jog movement in positive direction*)
		MoveJogNeg : BOOL; (*Starts the jog movement in negative direction*)
		ErrorAcknowledge : BOOL; (*Acknowledge an error with a pos. Edge*)
	END_STRUCT;
	Cyclic_Read_typ : 	STRUCT
		s_encoder : DINT;
		v_act : REAL;
		torq_act : REAL;
	END_STRUCT;
	Cyclic_Write_typ : 	STRUCT
		v_set : REAL;
		torq_set : REAL;
	END_STRUCT;
	MC_Axis_typ : 	STRUCT
		Step : UINT;
		AxisID : Axis_ID_typ; (*axis info*)
		AxisCmd : Axis_Cmd_typ; (*axis comdand*)
		Status : Axis_Status_typ;
		AxisState : Axis_State_typ;
		Parameter : Axis_Parameter_typ;
		CycRead : Cyclic_Read_typ;
		CycWrite : Cyclic_Write_typ;
		DriverStatus : MC_DRIVESTATUS_TYP; (*actual status of the axis*)
	END_STRUCT;
	Par_ID_typ : 	STRUCT
		ParID : UINT;
		DataType : UINT;
		DataAddress : UDINT;
		pValue : ARRAY[0..3]OF SINT;
	END_STRUCT;
	Par_RW_typ : 	STRUCT
		idxInit : UINT;
		idxWrite : UINT;
		idxRead : UINT;
		init : ARRAY[0..7]OF Par_ID_typ;
		Write : ARRAY[0..15]OF Par_ID_typ;
		Read : ARRAY[0..9]OF Par_ID_typ;
	END_STRUCT;
	Encoder_Par_typ : 	STRUCT
		count_dir : USINT; (*ENCOD_COUNT_DIR*)
		load_units : UDINT;
		encoder_rev : UDINT;
	END_STRUCT;
	Limit_Par_typ : 	STRUCT
		a1_pos : REAL;
		a2_pos : REAL;
		a1_neg : REAL;
		a2_neg : REAL;
		v_pos : REAL;
		v_neg : REAL;
	END_STRUCT;
	ParID_Read_typ : 	STRUCT
		torqueRated : REAL;
		currentRated : REAL;
		offset : REAL;
		actUDC : REAL;
		actCurrent : REAL;
		tempMotor : REAL;
		actLimitTorque : REAL;
		tempJunction : REAL;
		torqueMax : REAL;
	END_STRUCT;
	PID_Par_typ : 	STRUCT
		kv_p : REAL;
		tn_p : REAL;
		kv_s : REAL;
		tn_s : REAL;
		tf_s : REAL;
		kpJunction : REAL;
		kpMotorTemp : REAL;
		tdFF_s : REAL;
	END_STRUCT;
	Axis_Fix_typ : 	STRUCT
		encoderPar : Encoder_Par_typ;
		limitPar : Limit_Par_typ;
		pidPar : PID_Par_typ;
	END_STRUCT;
	ParID_Value_typ : 	STRUCT
		encoderPar : Encoder_Par_typ;
		limitPar : Limit_Par_typ;
		pidPar : PID_Par_typ;
		v_Max : REAL;
		readPar : ParID_Read_typ;
	END_STRUCT;
END_TYPE
```

#### Variables.var
```iecst
(*General Variables*)
VAR
	StepReadID : UINT := 0;
	StepWriteID : UINT := 0;
	FixTransferL : Axis_Fix_typ;
	mcAxis : MC_Axis_typ := (0);
	mcParID_RW : Par_RW_typ := (0);
	mcParID_Value : ParID_Value_typ := (0);
	mcDriverStatus : MC_DRIVESTATUS_TYP := (0);
	OldAlarmConfirmOK : USINT := 0;
	cmdStopPosOld : BOOL := 0;
	cmdMoveAbsolutePosOld : BOOL := 0;
END_VAR
(*Used Functionblocks*)
VAR
	MC_MoveVelocity_0 : MC_MoveVelocity; (*Function Block*)
	MC_Reset_0 : MC_Reset; (*Function Block*)
	MC_Home_0 : MC_Home; (*Function Block*)
	MC_Stop_0 : MC_Stop; (*Function Block*)
	MC_Power_0 : MC_Power; (*Function Block*)
	MC_ReadAxisError_0 : MC_ReadAxisError; (*Function Block*)
	MC_ReadStatus_0 : MC_ReadStatus; (*Function Block*)
	MC_MoveAdditive_0 : MC_MoveAdditive; (*Function Block*)
	MC_MoveAbsolute_0 : MC_MoveAbsolute; (*Function Block*)
	MC_Halt_0 : MC_Halt; (*Function Block*)
	MC_BR_ReadDriveStatus_0 : MC_BR_ReadDriveStatus; (*Function Block*)
	MC_BR_CyclicRead_0 : MC_BR_CyclicRead := (0); (*Function Block*)
	MC_BR_CyclicRead_1 : MC_BR_CyclicRead := (0); (*Function Block*)
	MC_BR_CyclicRead_2 : MC_BR_CyclicRead := (0); (*Function Block*)
	MC_BR_CyclicWrite_0 : MC_BR_CyclicWrite := (0); (*Function Block*)
	MC_BR_CyclicWrite_1 : MC_BR_CyclicWrite := (0); (*Function Block*)
	MC_BR_ReadParID_0 : MC_BR_ReadParID := (0); (*Function Block*)
	MC_BR_WriteParID_0 : MC_BR_WriteParID := (0); (*Function Block*)
	NegNetworkInit : USINT;
END_VAR
(*HWSwitch*)
VAR
	diNegHWSwitch : INT;
	diPosHWSwitch : INT;
END_VAR
```
